// TIA Portal project "Bancada" (V17)

(* hardware
DEVICE "S7-1200 station_1"  S7-1200 Station
   slot 0: "Rack_0"  S7-1200 Rack  Rack  V1.0
   slot 1: "PLC_1"  CPU 1212C AC/DC/Rly  6ES7 212-1BE40-0XB0  V4.5
DEVICE "GSD device_1"  GSD.Device.PN
   slot 0: "Rack"  Rack  V1.0
   slot 0: "danfoss-fc-series"  Danfoss FC PN  130B1135  V03.01.0
      slot 0: "Danfoss FC PN"  Danfoss FC PN
      slot 1: "Interface"  Interface
         slot 1: "Port 1"  Port 1
         slot 2: "Port 2"  Port 2
   slot 1: "PPO 4 - 6/6 Words, Danfoss Telegram 104_1"  PPO 4 - 6/6 Words, Danfoss Telegram 104
      slot 0: "Parameter Access Point"  Parameter Access Point
      slot 1: "PPO 4 - 6/6 Words, Danfoss Telegram 104"  PPO 4 - 6/6 Words, Danfoss Telegram 104
DEVICE "HMI_1"  KTP700 Basic PN
   slot 0: "HMI_1"  KTP700 Basic PN  6AV2 123-2GB03-0AX0  17.0.0.0
   slot 1: "HMI_RT_1"  KTP700 Basic PN  6AV2 123-2GB03-0AX0  17.0.0.0
   slot 5: "HMI_1.IE_CP_1"  PROFINET Interface  17.0.0.0
      slot 1: "PROFINET Interface_1"  PROFINET Interface
         slot 1: "Port_1"  Port
*)

// ===== PLC "PLC_1"  CPU 1212C AC/DC/Rly =====

VAR_GLOBAL   // PLC tag table "teste"
   "Tag_2" AT %M100.0 : Bool;
   "Tag_3" AT %MW300 : Int;
   "Tag_4" AT %MW302 : Int;
   "Tag_5" AT %MW306 : Int;
   "Tag_6" AT %MW308 : Int;
   "Tag_7" AT %MW304 : Int;
   "Tag_8" AT %MW310 : Int;
   "Tag_9" AT %MW312 : Int;
   "Tag_10" AT %MW314 : Int;
   "Tag_11" AT %MW316 : Int;
   "Tag_12" AT %MW320 : Int;
   "Tag_13" AT %MW318 : Int;
   "Tag_14" AT %MD400 : DWord;
   "Tag_15" AT %MD314 : Real;
   "Tag_16" AT %MD318 : Real;
   "Tag_17" AT %MD500 : DWord;
   "Tag_18" AT %MD504 : DWord;
END_VAR

VAR_GLOBAL   // PLC tag table "Default tag table"
   "DRV_EN_DUT1" AT %M0.0 : Bool;
   "RUN_DUT1" AT %M0.1 : Bool;
   "REVERSE_DUT1" AT %M0.2 : Bool;
   "RESET_DUT1" AT %M0.3 : Bool;
   "REF_VALUE_DUT1" AT %MW2 : Int;
   "READY_DUT1" AT %M0.4 : Bool;
   "FAULT_DUT1" AT %M0.5 : Bool;
   "WARNING_DUT1" AT %M0.6 : Bool;
   "RUNNING_DUT1" AT %M0.7 : Bool;
   "RUN_ON_REF_DUT1" AT %M1.0 : Bool;
   "MAV_DUT1" AT %MW4 : Int;
   "MOTORCURRENT_DUT1" AT %MD6 : Real;
   "COMM_ERR_DUT1" AT %MW10 : Int;
   "EXECUTE_DUT1" AT %M1.1 : Bool;
   "RD_WR_DUT1" AT %M1.2 : Bool;
   "PAR_NO_DUT1" AT %MW12 : Word;
   "INDEX_DUT1" AT %MW14 : Word;
   "WR_VALUE_DUT1" AT %MD16 : DWord;
   "BUSY_DUT1" AT %M1.3 : Bool;
   "DONE_DUT1" AT %M1.4 : Bool;
   "FAULT_PARA_DUT1" AT %M1.5 : Bool;
   "RD_VALUE_DUT1" AT %MD20 : DWord;
   "FALUT_CODE_DUT1" AT %MD24 : DWord;
   "CH_ERR_TYP_DUT1" AT %MW28 : Word;
   "ALARM_DUT1" AT %MD30 : DWord;
   "DIAG_WARNING_DUT1" AT %MD34 : DWord;
   "DIAG_ALARM_DUT1" AT %MD38 : DWord;
   "Test" AT %M1.6 : Bool;
   "FB_CTRL_EN_DUT1" AT %M1.7 : Bool;
   "COMM_ERR_FLEXIBLE_DUT1" AT %MW42 : Int;
   "START_FLEXIBLE_CTRL_DUT1" AT %M44.0 : Bool;
   "REF_VALUE_FLEXI_CTRL_DUT1" AT %MW46 : Int;
   "Tag_1" AT %M300.0 : Bool;
   "DC_BRAKE_RAMP" AT %M44.1 : Bool;
   "test1" AT %M44.2 : Bool;
   "Dummy" AT %M44.3 : Bool;
   "PRESET_REF1_DUT1" AT %M44.4 : Bool;
   "PRESET_REF2_DUT1" AT %M44.5 : Bool;
   "DC_BRAKE_RAMP_DUT1" AT %M44.6 : Bool;
   "COAST_INV_DUT1" AT %M44.7 : Bool;
   "QSTP_RMP_DUT1" AT %M45.0 : Bool;
   "HLD_RAMP_DUT1" AT %M45.1 : Bool;
   "RESET_DUT_FLEXIBLE_CTRL_DUT1" AT %M45.2 : Bool;
   "JOG_DUT1" AT %M45.3 : Bool;
   "RAMP_1_2_DUT1" AT %M45.4 : Bool;
   "RLY_1_NO_DUT1" AT %M45.5 : Bool;
   "RLY_2_ON_DUT1" AT %M45.6 : Bool;
   "SETUP_SEL_1_DUT1" AT %M45.7 : Bool;
   "SETUP_SEL_2_DUT1" AT %M48.0 : Bool;
   "REVERSE_FLEXIBLE_CTRl_DUT1" AT %M48.1 : Bool;
   "READ_FLEXIBLE_CTRL_DUT1" AT %M48.2 : Bool;
   "FALUT_FLEXIBLE_CTRL_DUT1" AT %M48.3 : Bool;
   "WARNING_FLEXIBLE_CTRL_DUT1" AT %M48.4 : Bool;
   "RUN_ON_REF_FLEXIBLE_CTRL_DUT1" AT %M48.5 : Bool;
   "RUNNING_FLEXIBLE_CTRL_DUT1" AT %M48.6 : Bool;
   "MAV_FLEXIBLE_CTRL_DUT1" AT %MW50 : Int;
   "EN_BASIC" AT %M48.7 : Bool;
   "EN_FLEXIBLE_CTRL" AT %M49.0 : Bool;
   "EN_FLEXIBLE" AT %M49.1 : Bool;
   "EN_PARAM_ACCESS" AT %M49.2 : Bool;
   "EN_DIAGNOSTICS" AT %M49.3 : Bool;
   "DRV_EN_DUT2" AT %M49.4 : Bool;
   "RUN_DUT2" AT %M49.5 : Bool;
   "REVERSE_DUT2" AT %M49.6 : Bool;
   "RESET_DUT2" AT %M49.7 : Bool;
   "REF_VALUE_DUT2" AT %MW52 : Int;
   "READY_DUT2" AT %M54.0 : Bool;
   "FAULT_DUT2" AT %M54.1 : Bool;
   "WARNING_DUT2" AT %M54.2 : Bool;
   "RUNNING_DUT2" AT %M54.3 : Bool;
   "RUN_ON_REF_DUT2" AT %M54.4 : Bool;
   "MAV_DUT2" AT %MW56 : Int;
   "MOTORCURRENT_DUT2" AT %MD58 : Real;
   "COMM_ERR_DUT2" AT %MW62 : Int;
   "PRESET_REF1_DUT2" AT %M54.5 : Bool;
   "PRESET_REF2_DUT2" AT %M54.6 : Bool;
   "DC_BRAKE_RAMP_DUT2" AT %M54.7 : Bool;
   "COAST_INV_DUT2" AT %M55.0 : Bool;
   "QSTP_RMP_DUT2" AT %M55.1 : Bool;
   "HLD_RAMP_DUT2" AT %M55.2 : Bool;
   "START_FLEXIBLE_CTRL_DUT2" AT %M55.3 : Bool;
   "RESET_DUT_FLEXIBLE_CTRL_DUT2" AT %M55.4 : Bool;
   "JOG_DUT2" AT %M55.5 : Bool;
   "RAMP_1_2_DUT2" AT %M55.6 : Bool;
   "RLY_1_NO_DUT2" AT %M55.7 : Bool;
   "RLY_2_ON_DUT2" AT %M64.0 : Bool;
   "SETUP_SEL_1_DUT2" AT %M64.1 : Bool;
   "SETUP_SEL_2_DUT2" AT %M64.2 : Bool;
   "REVERSE_FLEXIBLE_CTRl_DUT2" AT %M64.3 : Bool;
   "REF_VALUE_FLEXI_CTRL_DUT2" AT %MW66 : Int;
   "READ_FLEXIBLE_CTRL_DUT2" AT %M64.4 : Bool;
   "FALUT_FLEXIBLE_CTRL_DUT2" AT %M64.5 : Bool;
   "WARNING_FLEXIBLE_CTRL_DUT2" AT %M64.6 : Bool;
   "RUNNING_FLEXIBLE_CTRL_DUT2" AT %M64.7 : Bool;
   "MAV_FLEXIBLE_CTRL_DUT2" AT %MW68 : Int;
   "RUN_ON_REF_FLEXIBLE_CTRL_DUT2" AT %M65.0 : Bool;
   "FB_CTRL_EN_DUT2" AT %M65.1 : Bool;
   "COMM_ERR_FLEXIBLE_DUT2" AT %MW70 : Int;
   "DATA_VALID_DUT1" AT %M65.2 : Bool;
   "DATA_VALID_DUT2" AT %M65.3 : Bool;
   "EXECUTE_DUT2" AT %M65.4 : Bool;
   "RD_WR_DUT2" AT %M65.5 : Bool;
   "PAR_NO_DUT2" AT %MW72 : Word;
   "INDEX_DUT2" AT %MW74 : Word;
   "WR_VALUE_DUT2" AT %MD76 : DWord;
   "BUSY_DUT2" AT %M65.6 : Bool;
   "DONE_DUT2" AT %M65.7 : Bool;
   "FAULT_PARA_DUT2" AT %M80.0 : Bool;
   "RD_VALUE_DUT2" AT %MD82 : DWord;
   "FALUT_CODE_DUT2" AT %MD86 : DWord;
   "ALARM_1_DUT1" AT %MD90 : DWord;
   "WARNING_1_DUT1" AT %MD94 : DWord;
   "CH_ERR_TYP_DUT2" AT %MW98 : Word;
   "ALARM_1_DUT2" AT %MD100 : DWord;
   "WARNING_1_DUT2" AT %MD104 : DWord;
END_VAR

VAR_GLOBAL CONSTANT   // PLC tag table "Default tag table"
   "None(1)" : Pip := 65535;
   "Automatic update(1)" : Pip := 0;
   "PIP 1(1)" : Pip := 1;
   "PIP 2(1)" : Pip := 2;
   "PIP 3(1)" : Pip := 3;
   "PIP 4(1)" : Pip := 4;
   "PIP 5" : Pip := 5;
   "PIP 6" : Pip := 6;
   "PIP 7" : Pip := 7;
   "PIP 8" : Pip := 8;
   "PIP 9" : Pip := 9;
   "PIP 10" : Pip := 10;
   "PIP 11" : Pip := 11;
   "PIP 12" : Pip := 12;
   "PIP 13" : Pip := 13;
   "PIP 14" : Pip := 14;
   "PIP 15" : Pip := 15;
   "PIP 16" : Pip := 16;
   "PIP 17" : Pip := 17;
   "PIP 18" : Pip := 18;
   "PIP 19" : Pip := 19;
   "PIP 20" : Pip := 20;
   "PIP 21" : Pip := 21;
   "PIP 22" : Pip := 22;
   "PIP 23" : Pip := 23;
   "PIP 24" : Pip := 24;
   "PIP 25" : Pip := 25;
   "PIP 26" : Pip := 26;
   "PIP 27" : Pip := 27;
   "PIP 28" : Pip := 28;
   "PIP 29" : Pip := 29;
   "PIP 30" : Pip := 30;
   "PIP 31" : Pip := 31;
   "PIP OB Servo(1)" : Pip := 32768;
   "Local~MC(1)" : Hw_SubModule := 51;
   "Local~Display" : Hw_SubModule := 54;
   "Local~Exec(1)" : Hw_SubModule := 52;
   "Local(1)" : Hw_SubModule := 49;
   "Local~DP_interface_1" : Hw_Interface := 60;
   "Local~PROFINET_interface_1(1)" : Hw_Interface := 64;
   "Local~PROFINET_interface_1~Port_1(1)" : Hw_Interface := 65;
   "Local~PROFINET_interface_1~Port_2" : Hw_Interface := 66;
   "Local~PROFINET_interface_2" : Hw_Interface := 72;
   "Local~PROFINET_interface_2~Port_1" : Hw_Interface := 73;
   "OB_Main(1)" : OB_PCYCLE := 1;
   "Local~PROFINET_IO-System" : Hw_IoSystem := 257;
   "OB_Diagnostic error interrupt" : OB_DIAG := 82;
   "Local~DP-Mastersystem" : Hw_IoSystem := 268;
   "profinetdut1~Proxy" : Hw_SubModule := 258;
   "profinetdut1~IODevice" : Hw_Device := 263;
   "profinetdut1~Interface" : Hw_Interface := 259;
   "profinetdut1~Interface~Port_1" : Hw_Interface := 260;
   "profinetdut1~Interface~Port_2" : Hw_Interface := 261;
   "profinetdut1~Head" : Hw_SubModule := 262;
   "profinetdut2~Proxy" : Hw_SubModule := 271;
   "profinetdut2~IODevice" : Hw_Device := 269;
   "profinetdut2~Interface" : Hw_Interface := 272;
   "profinetdut2~Interface~Port_1" : Hw_Interface := 273;
   "profinetdut2~Interface~Port_2" : Hw_Interface := 274;
   "profinetdut2~Head" : Hw_SubModule := 275;
   "Slave_1~Head" : Hw_Interface := 281;
   "Slave_1~DPSlave" : Hw_DpSlave := 279;
   "Slave_1~PPO_Type_2_Module_consistent_PCD_2_1" : Hw_SubModule := 282;
   "Slave_1~PPO_Type_2_Module_consistent_PCD_2_2" : Hw_SubModule := 283;
   "profinetdut1~PPO_4_-_6_6_Words__Danfoss_Telegram,,," : Hw_SubModule := 265;
   "profinetdut1~PPO_4_-_6_6_Words__Danfoss_Telegra,,,~Parameter_Access_Point" : Hw_SubModule := 266;
   "profinetdut1~PPO_4_-_6_6_Words__Danfoss_Telegra,,,~PPO_4_-_6_6_Words__Danfoss_,,," : Hw_SubModule := 267;
   "profinetdut2~PPO_8_-_10_10_Words__Danfoss_Telegr,,," : Hw_SubModule := 276;
   "profinetdut2~PPO_8_-_10_10_Words__Danfoss_Teleg,,,~Parameter_Access_Point" : Hw_SubModule := 277;
   "profinetdut2~PPO_8_-_10_10_Words__Danfoss_Teleg,,,~PPO_8_-_10_10_Words__Danfos,,," : Hw_SubModule := 278;
   "Local~Common(1)" : Hw_SubModule := 50;
   "Local~Device(1)" : Hw_Device := 32;
   "Local~Configuration(1)" : Hw_SubModule := 33;
   "Local~License_Manager" : Hw_SubModule := 42;
   "Local~Virtual_communication_interface" : Hw_Interface := 135;
END_VAR

TYPE "PPO_READ_FCPROFILE"
TITLE = PPO_READ_FCPROFILE
// User defined data tyoe of input data read structure . Holds the data structure obtained from the Process data (PCDREAD) expressed in user data accessible format user
   STRUCT
      STW : Struct   // Status word
         BIT_00_CTRL_RDY : Bool;   // 0=Control not ready, 1=Control ready
         BIT_01_DRV_RDY : Bool;   // 0=Frequency converter, 1=Frequency converter ready
         BIT_02_COAST_RDY : Bool;   // 0=Coasting, 1=Enable
         BIT_03_TRIP : Bool;   // 0=No error, 1=Trip
         BIT_04_ERROR : Bool;   // 0=No error, 1=Error (no trip)
         BIT_05_RESERVED : Bool;   // 0=Reserved, 1=---
         BIT_06_TRIPLOCK : Bool;   // 0=No error, 1=Triplock
         BIT_07_WARNING : Bool;   // 0=No warning, 1=Warning
         BIT_08_RUNNING_REF : Bool;   // 0=Speed <> reference, 1=Speed=reference
         BIT_09_CTRL_SOURCE : Bool;   // 0=Local operation, 1=Bus control
         BIT_10_F_LIMIT_OK : Bool;   // 0=Out of frequency limit, 1=Frequency limit ok
         BIT_11_IN_OPR : Bool;   // 0=No operation, 1=In operation
         BIT_12_IN_AUTOSTART : Bool;   // 0=Frequency converter OK, 1=Stopped, autostart
         BIT_13_VOLT_MAX : Bool;   // 0=Voltage OK, 1=Voltage exceeded
         BIT_14_TORQ_MAX : Bool;   // 0=Torque OK, 1=Torque exceeded
         BIT_15_TIMER_EXD : Bool;   // 0=Timer OK, 1=Timer exceeded
      END_STRUCT;
      MAV : Int;   // Measured Actual Value (Speed) in raw value (-16384) to (+16384)
      PCD_02 : Int;   // Depends on Drive config.
      PCD_03 : Int;   // Depends on Drive config.
      PCD_04 : Int;   // Depends on Drive config.
      PCD_05 : Int;   // Depends on Drive config.
      PCD_06 : Int;   // Depends on Drive config.
      PCD_07 : Int;   // Depends on Drive config.
      PCD_08 : Int;   // Depends on Drive config.
      PCD_09 : Int;   // Depends on Drive config.
   END_STRUCT;
END_TYPE

TYPE "PPO_WRITE_FCPROFILE"
TITLE = PPO_WRITE_FCPROFILE
// User defined data type of input data read structure. Holds the data structure obtained from the Process data(PCDWRITE) expressed in user data accessible format user
   STRUCT
      CTW : Struct   // Control word
         BIT_00_PRESET_REF_1 : Bool;   // 0=Reference value, 1=selection lsb
         BIT_01_PRESET_REF_2 : Bool;   // 0=Reference value, 1=selection msb
         BIT_02_DC_BRAKE_RAMP : Bool := TRUE;   // 0=DC brake, 1=Ramp
         BIT_03_COAST_INV : Bool := TRUE;   // 0=Coasting, 1=No coasting
         BIT_04_QSTP_RMP : Bool := TRUE;   // 0=Quick stop, 1=Ramp
         BIT_05_HLD_RMP : Bool := TRUE;   // 0=Hold output frequency, 1=Use ramp
         BIT_06_START : Bool;   // 0=Ramp stop, 1=Start
         BIT_07_RESET : Bool;   // 0=No function, 1=Reset
         BIT_08_JOG : Bool;   // 0=No function, 1=Jog
         BIT_09_RAMP_1_2 : Bool;   // 0=Ramp 1, 1=Ramp 2
         BIT_10_DATA_VALID : Bool := TRUE;   // 0=Dont use CTW, 1= Use CTW
         BIT_11_RLY_1_ON : Bool := FALSE;   // 0=Relay 01 deactived, 1=Relay 01 active
         BIT_12_RLY_2_ON : Bool := FALSE;   // 0=Relay 02 deactived, 1=Relay 02 active
         BIT_13_SETUP_SEL_1 : Bool := FALSE;   // 0=Parameter set-up, 1=selection lsb
         BIT_14_SETUP_SEL_2 : Bool := FALSE;   // 0=Parameter set-up, 1=selection msb
         BIT_15_REVERSE : Bool;   // 0= No Reverse, 1= Reverse
      END_STRUCT;
      REF_VALUE : Int;   // Main Ref. value (Speed) in raw value. (-16384) to (+16384)
      PCD_02 : Int;   // Depends on Drive config.
      PCD_03 : Int;   // Depends on Drive config.
      PCD_04 : Int;   // Depends on Drive config.
      PCD_05 : Int;   // Depends on Drive config.
      PCD_06 : Int;   // Depends on Drive config.
      PCD_07 : Int;   // Depends on Drive config.
      PCD_08 : Int;   // Depends on Drive config.
      PCD_09 : Int;   // Depends on Drive config.
   END_STRUCT;
END_TYPE

TYPE "PPO_READ_PROFIDRIVE_PROFILE"
   STRUCT
      STW : Struct   // Status word
         BIT_08_RUNNING_REF : Bool;   // 0=Speed <> reference, 1=Speed=reference
         BIT_09_CTRL_SOURCE : Bool;   // 0=Local operation, 1=Bus control
         BIT_10_F_LIMIT_OK : Bool;   // 0=Out of frequency limit, 1=Frequency limit ok
         BIT_11 : Bool;   // Device specific
         BIT_12_IN_AUTOSTART : Bool;   // 0=Frequency converter OK, 1=Stopped, autostart
         BIT_13_DRV_RDY : Bool;   // 0=Drive is not ready, 1=Drive is ready to go to running state
         BIT_14 : Bool;   // ???
         BIT_15 : Bool;   // ???
         BIT_00_CTRL_RDY : Bool;   // 0=Control not ready, 1=Control ready
         BIT_00_RDY_TO_OPR : Bool;   // 0=Not Ready To Operate, 1=Ready To Operate
         BIT_02_OPR_EN : Bool;   // 0=Operation Disabled, 1=Operation Enabled
         BIT_03_FAULT : Bool;   // 0=No Fault, 1=Fault
         BIT_04_COAST_STP : Bool;   // 0=Coast Stop Activated, 1=Coast Stop not Activated
         BIT_05_QUICK_STP : Bool;   // 0=Quick Stop Not Activated, 1=Quick Stop Activated
         BIT_06_SWTCH_ON_INH : Bool;   // 0=Switching On Not Inhibited, 1=Switching On Inhibited
         BIT_07_WARNING : Bool;   // 0=No warning, 1=Warning
      END_STRUCT;
      MAV : Int;   // Main actual value (Speed) in %
      PCD_02 : Int;   // Depends on Drive config.
      PCD_03 : Int;   // Depends on Drive config.
      PCD_04 : Int;   // Depends on Drive config.
      PCD_05 : Int;   // Depends on Drive config.
      PCD_06 : Int;   // Depends on Drive config.
      PCD_07 : Int;   // Depends on Drive config.
      PCD_08 : Int;   // Depends on Drive config.
      PCD_09 : Int;   // Depends on Drive config.
      PCD_11 : Int;   // Depends on Drive config.
   END_STRUCT;
END_TYPE

TYPE "PPO_WRITE_PROFIDRIVE_PROFILE"
   STRUCT
      CTW : Struct   // Control word
         BIT_08_NOTUSED : Bool;   // Not used
         BIT_09_NOTUSED : Bool;   // Not used
         BIT_10_USE_CTRL_WORD : Bool := TRUE;   // 0=No Control by PLC, 1=Control by PLC
         BIT_11_DEV_SPEC : Bool := FALSE;   // Device specific
         BIT_12_DEV_SPEC : Bool := FALSE;   // Device specific
         BIT_13_DEV_SPEC : Bool := FALSE;   // Device specific
         BIT_14_DEV_SPEC : Bool := FALSE;   // Device specific
         BIT_15_DEV_SPEC : Bool;   // Device specific
         BIT_00_ON_1 : Bool;   // 0=Control not ready, 1=Control ready
         BIT_01_COAST_INV : Bool;   // 0=Coast Stop, 1=No Coast Stop
         BIT_02_QUICK_INV : Bool := TRUE;   // 0=Quick Stop, 1=No Quick Stop
         BIT_03_EN_OPR : Bool := TRUE;   // 0=Operation disabled, 1=Operation enabled
         BIT_04_RAMP : Bool := TRUE;   // 0=Reset Ramp Generator, 1=Enable Ramp Generator
         BIT_05_USE_RAMP : Bool := TRUE;   // 0=Freeze Ramp Generator, 1=Unfreeze Ramp Generator
         BIT_06_START : Bool;   // 0=Disable Set Point, 1=Enable Setpoint
         BIT_07_RESET_ERR : Bool;   // 0=No Reset, 1=Reset Fault, rising edge
      END_STRUCT;
      MRV : Int;   // Main Ref. value (Speed) in %
      PCD_02 : Word;   // Depends on Drive config.
      PCD_03 : Word;   // Depends on Drive config.
      PCD_04 : Word;   // Depends on Drive config.
      PCD_05 : Word;   // Depends on Drive config.
      PCD_06 : Word;   // Depends on Drive config.
      PCD_07 : Word;   // Depends on Drive config.
      PCD_08 : Word;   // Depends on Drive config.
      PCD_09 : Word;   // Depends on Drive config.
      PCD_10 : Word;   // Depends on Drive config.
   END_STRUCT;
END_TYPE

TYPE "PPO_DRIVEPROFILE"
   STRUCT
      PPO_PD : Struct
         RD : "PPO_READ_PROFIDRIVE_PROFILE";
         WR : "PPO_WRITE_PROFIDRIVE_PROFILE";
      END_STRUCT;
   END_STRUCT;
END_TYPE

TYPE "PPO_FC"
TITLE = PPO_FC
// User defined data type of Input data read structure and output data write structure. Holds the data structure obtained from the Process data (PCDREAD) and (PCDWRITE) expressed in user data accessible format user
   STRUCT
      PPO_FC : Struct
         RD : "PPO_READ_FCPROFILE";
         WR : "PPO_WRITE_FCPROFILE";
      END_STRUCT;
   END_STRUCT;
END_TYPE

TYPE "PCD"
   STRUCT
      PCD : Struct
         PCDREAD : "PPO_READ_FCPROFILE";
         PCDWRITE : "PPO_WRITE_FCPROFILE";
      END_STRUCT;
   END_STRUCT;
END_TYPE

DATA_BLOCK "VLT_PROFI_FC_DIAGNOSTICS_DB_2"   // DB1
{ S7_Optimized_Access := 'TRUE' }
AUTHOR : Danfoss_Drives
FAMILY : VLT
VERSION : 1.12
// stored: InstanceOfName VLT_PROFI_FC_DIAGNOSTICS
"VLT_PROFI_FC_DIAGNOSTICS"
BEGIN
END_DATA_BLOCK

DATA_BLOCK "VLT_PROFI_FC_PARAM_ACCESS_DB"   // DB2
{ S7_Optimized_Access := 'FALSE' }
AUTHOR : Danfoss
FAMILY : VLT
VERSION : 1.0
// stored: InstanceOfName VLT_PROFI_FC_PARAM_ACCESS
"VLT_PROFI_FC_PARAM_ACCESS"
BEGIN
END_DATA_BLOCK

DATA_BLOCK "VLT_PROFI_FC_DIAGNOSTICS_DB"   // DB3
{ S7_Optimized_Access := 'TRUE' }
AUTHOR : Danfoss
FAMILY : VLT
VERSION : 1.0
// stored: InstanceOfName VLT_PROFI_FC_DIAGNOSTICS
"VLT_PROFI_FC_DIAGNOSTICS"
BEGIN
END_DATA_BLOCK

DATA_BLOCK "VLT_PROFI_FC_FLEXIBLE_CTRL_DB"   // DB5
{ S7_Optimized_Access := 'TRUE' }
AUTHOR : Danfoss
FAMILY : VLT
VERSION : 1.0
// stored: InstanceOfName VLT_PROFI_FC_FLEXIBLE_CTRL
"VLT_PROFI_FC_FLEXIBLE_CTRL"
BEGIN
END_DATA_BLOCK

DATA_BLOCK "VLT_PROFI_FC_PARAM_ACCESS_DB_1"   // DB6
{ S7_Optimized_Access := 'FALSE' }
AUTHOR : Danfoss
FAMILY : VLT
VERSION : 1.0
// stored: InstanceOfName VLT_PROFI_FC_PARAM_ACCESS
"VLT_PROFI_FC_PARAM_ACCESS"
BEGIN
END_DATA_BLOCK

DATA_BLOCK "VLT_PROFI_FC_DIAGNOSTICS_DB_1"   // DB7
{ S7_Optimized_Access := 'TRUE' }
AUTHOR : Danfoss
FAMILY : VLT
VERSION : 1.0
// stored: InstanceOfName VLT_PROFI_FC_DIAGNOSTICS
"VLT_PROFI_FC_DIAGNOSTICS"
BEGIN
END_DATA_BLOCK

DATA_BLOCK "VLT_PROFI_FC_FLEXIBLE_CTRL_DB_1"   // DB8
{ S7_Optimized_Access := 'TRUE' }
AUTHOR : Danfoss
FAMILY : VLT
VERSION : 1.0
// stored: InstanceOfName VLT_PROFI_FC_FLEXIBLE_CTRL
"VLT_PROFI_FC_FLEXIBLE_CTRL"
BEGIN
END_DATA_BLOCK

DATA_BLOCK "data"   // DB9
{ S7_Optimized_Access := 'TRUE' }
VERSION : 0.1
   VAR
      Input2 : Int;
      Input : Int;
   END_VAR
BEGIN
END_DATA_BLOCK

DATA_BLOCK "db2"   // DB10
{ S7_Optimized_Access := 'TRUE' }
VERSION : 0.1
// stored: InstanceOfName web
"web"
BEGIN
END_DATA_BLOCK

DATA_BLOCK "date"   // DB11
{ S7_Optimized_Access := 'TRUE' }
VERSION : 0.1
   VAR
      in : Int;
      corrente : Real;
      frequencia : Real;
      start : Bool;
      reset : Bool;
      reversao : Bool;
      jog : Bool;
   END_VAR
BEGIN
END_DATA_BLOCK

// folder: VLT_PROFI_LIB_V1_12

DATA_BLOCK "VLT_PCD_DATA"   // DB100
TITLE = VLT_PCD_DATA
{ S7_Optimized_Access := 'TRUE' }
AUTHOR : Danfoss_Drives
FAMILY : VLT
VERSION : 1.12
// Data block of input data read structure and output data write structure. Holds the data structure obtained from the Process data (PCDREAD) and (PCDWRITE) expressed in user data accessible format user
   VAR
      VLT_PCD_DATA : Array[0..10] of "PPO_FC";
   END_VAR
BEGIN
END_DATA_BLOCK

// folder: (top level)

FUNCTION_BLOCK "web"   // FB1, LAD
{ S7_Optimized_Access := 'TRUE' }
VERSION : 0.1
   VAR
      timer1 : TON_TIME;
      timer2 : TON_TIME;
   END_VAR
BEGIN

REGION Network 1
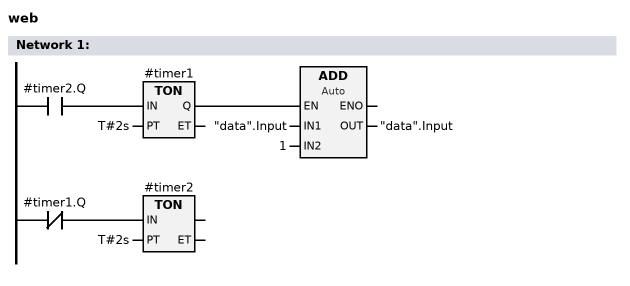
   #timer1(IN := #timer2.Q, PT := T#2s);   // TON
   IF #timer1.Q THEN "data".Input := "data".Input + 1; END_IF;
   #timer2(IN := NOT #timer1.Q, PT := T#2s);   // TON
END_REGION
END_FUNCTION_BLOCK

ORGANIZATION_BLOCK "Main"   // OB1, LAD, ProgramCycle
TITLE = "Main Program Sweep (Cycle)"
{ S7_Optimized_Access := 'TRUE' }
VERSION : 0.1
   VAR_INPUT
      Initial_Call : Bool;   // Initial call of this OB
      Remanence : Bool;   // =True, if remanent data are available
   END_VAR
   VAR_TEMP
      erro : Int;
   END_VAR
   VAR_TEMP   // added for the SCL form of the ladder/FBD networks
      _w1 : Bool;
   END_VAR
BEGIN

REGION Network 1
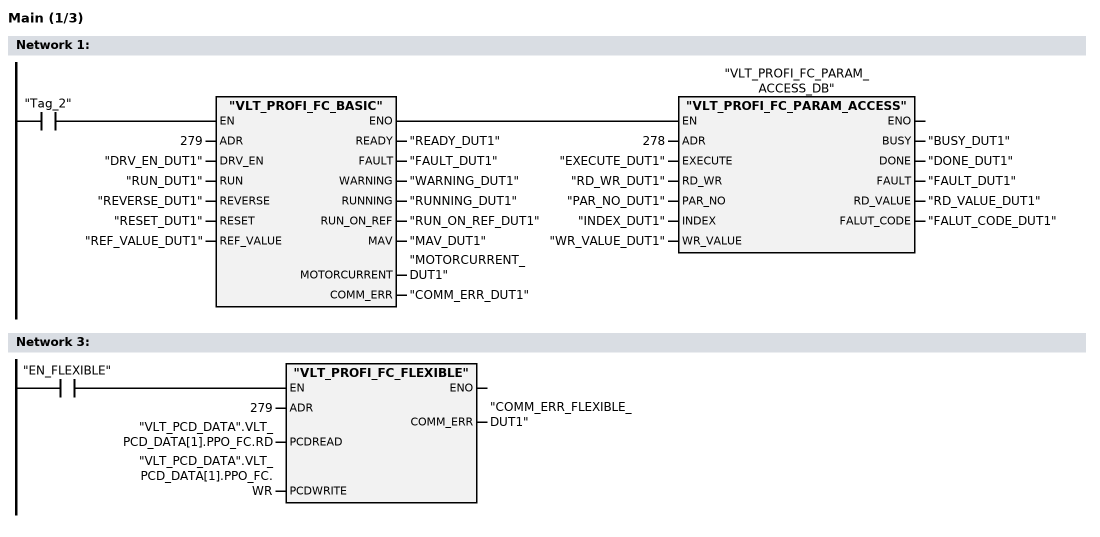
   RUNG wire#powerrail
      Contact( "Tag_2" )
      "VLT_PROFI_FC_BASIC"(ADR := 279, DRV_EN := "DRV_EN_DUT1", RUN := "RUN_DUT1", REVERSE := "REVERSE_DUT1", RESET := "RESET_DUT1", REF_VALUE := "REF_VALUE_DUT1", READY => "READY_DUT1", FAULT => "FAULT_DUT1", WARNING => "WARNING_DUT1", RUNNING => "RUNNING_DUT1", RUN_ON_REF => "RUN_ON_REF_DUT1", MAV => "MAV_DUT1", MOTORCURRENT => "MOTORCURRENT_DUT1", COMM_ERR => "COMM_ERR_DUT1")
      "VLT_PROFI_FC_PARAM_ACCESS_DB"(ADR := 278, EXECUTE := "EXECUTE_DUT1", RD_WR := "RD_WR_DUT1", PAR_NO := "PAR_NO_DUT1", INDEX := "INDEX_DUT1", WR_VALUE := "WR_VALUE_DUT1", BUSY => "BUSY_DUT1", DONE => "DONE_DUT1", FAULT => "FAULT_DUT1", RD_VALUE => "RD_VALUE_DUT1", FALUT_CODE => "FALUT_CODE_DUT1")
   END_RUNG
   // the same network as SCL:
   "VLT_PROFI_FC_BASIC"(EN := "Tag_2",
                        ADR := 279,
                        DRV_EN := "DRV_EN_DUT1",
                        RUN := "RUN_DUT1",
                        REVERSE := "REVERSE_DUT1",
                        RESET := "RESET_DUT1",
                        REF_VALUE := "REF_VALUE_DUT1",
                        READY => "READY_DUT1",
                        FAULT => "FAULT_DUT1",
                        WARNING => "WARNING_DUT1",
                        RUNNING => "RUNNING_DUT1",
                        RUN_ON_REF => "RUN_ON_REF_DUT1",
                        MAV => "MAV_DUT1",
                        MOTORCURRENT => "MOTORCURRENT_DUT1",
                        COMM_ERR => "COMM_ERR_DUT1",
                        ENO => #_w1);
   IF #_w1 THEN
       "VLT_PROFI_FC_PARAM_ACCESS_DB"(ADR := 278,   // "VLT_PROFI_FC_PARAM_ACCESS"
                               EXECUTE := "EXECUTE_DUT1",
                               RD_WR := "RD_WR_DUT1",
                               PAR_NO := "PAR_NO_DUT1",
                               INDEX := "INDEX_DUT1",
                               WR_VALUE := "WR_VALUE_DUT1",
                               BUSY => "BUSY_DUT1",
                               DONE => "DONE_DUT1",
                               FAULT => "FAULT_DUT1",
                               RD_VALUE => "RD_VALUE_DUT1",
                               FALUT_CODE => "FALUT_CODE_DUT1");
   END_IF;
END_REGION

REGION Network 3
   RUNG wire#powerrail
      Contact( "EN_FLEXIBLE" )
      "VLT_PROFI_FC_FLEXIBLE"(ADR := 279, PCDREAD := "VLT_PCD_DATA".VLT_PCD_DATA[1].PPO_FC.RD, PCDWRITE := "VLT_PCD_DATA".VLT_PCD_DATA[1].PPO_FC.WR, COMM_ERR => "COMM_ERR_FLEXIBLE_DUT1")
   END_RUNG
   // the same network as SCL:
   IF "EN_FLEXIBLE" THEN
       "VLT_PROFI_FC_FLEXIBLE"(ADR := 279,
                               PCDREAD := "VLT_PCD_DATA".VLT_PCD_DATA[1].PPO_FC.RD,
                               PCDWRITE := "VLT_PCD_DATA".VLT_PCD_DATA[1].PPO_FC.WR,
                               COMM_ERR => "COMM_ERR_FLEXIBLE_DUT1");
   END_IF;
END_REGION

REGION Network 4
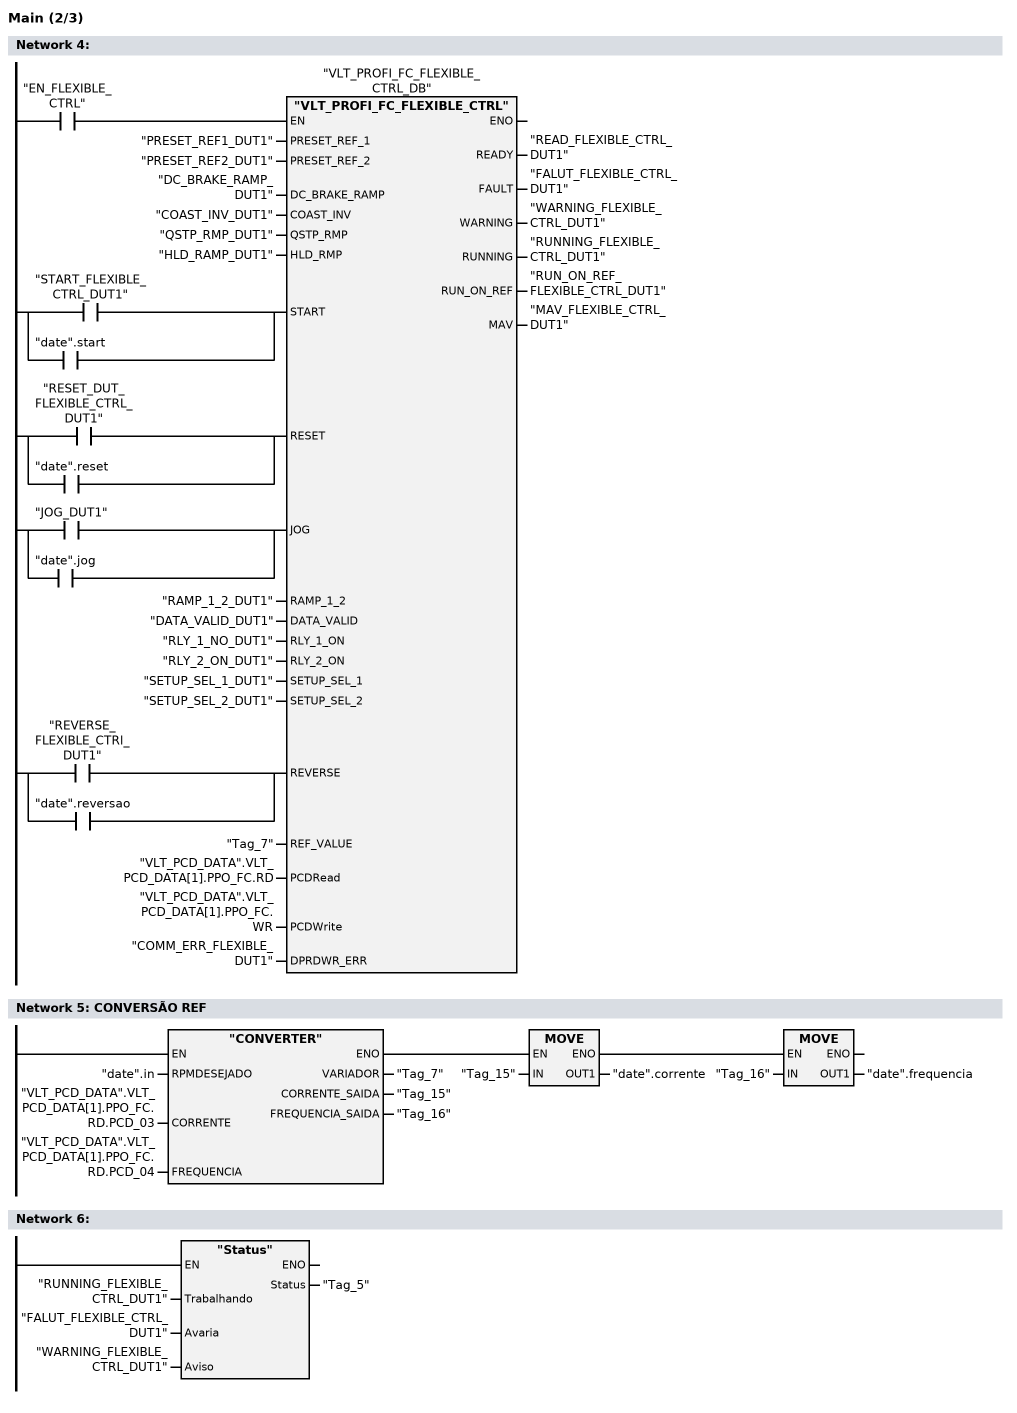
   RUNG wire#powerrail
      Contact( "EN_FLEXIBLE_CTRL" )
      "VLT_PROFI_FC_FLEXIBLE_CTRL_DB"(START := wire#w1, RESET := wire#w2, JOG := wire#w3, REVERSE := wire#w4, PRESET_REF_1 := "PRESET_REF1_DUT1", PRESET_REF_2 := "PRESET_REF2_DUT1", DC_BRAKE_RAMP := "DC_BRAKE_RAMP_DUT1", COAST_INV := "COAST_INV_DUT1", QSTP_RMP := "QSTP_RMP_DUT1", HLD_RMP := "HLD_RAMP_DUT1", RAMP_1_2 := "RAMP_1_2_DUT1", DATA_VALID := "DATA_VALID_DUT1", RLY_1_ON := "RLY_1_NO_DUT1", RLY_2_ON := "RLY_2_ON_DUT1", SETUP_SEL_1 := "SETUP_SEL_1_DUT1", SETUP_SEL_2 := "SETUP_SEL_2_DUT1", REF_VALUE := "Tag_7", PCDRead := "VLT_PCD_DATA".VLT_PCD_DATA[1].PPO_FC.RD, PCDWrite := "VLT_PCD_DATA".VLT_PCD_DATA[1].PPO_FC.WR, DPRDWR_ERR := "COMM_ERR_FLEXIBLE_DUT1", READY => "READ_FLEXIBLE_CTRL_DUT1", FAULT => "FALUT_FLEXIBLE_CTRL_DUT1", WARNING => "WARNING_FLEXIBLE_CTRL_DUT1", RUNNING => "RUNNING_FLEXIBLE_CTRL_DUT1", RUN_ON_REF => "RUN_ON_REF_FLEXIBLE_CTRL_DUT1", MAV => "MAV_FLEXIBLE_CTRL_DUT1")
   END_RUNG
   RUNG wire#powerrail
      Contact( "START_FLEXIBLE_CTRL_DUT1" )
   END_RUNG wire#w1
   RUNG wire#powerrail
      Contact( "date".start )
   END_RUNG wire#w1
   RUNG wire#powerrail
      Contact( "RESET_DUT_FLEXIBLE_CTRL_DUT1" )
   END_RUNG wire#w2
   RUNG wire#powerrail
      Contact( "date".reset )
   END_RUNG wire#w2
   RUNG wire#powerrail
      Contact( "JOG_DUT1" )
   END_RUNG wire#w3
   RUNG wire#powerrail
      Contact( "date".jog )
   END_RUNG wire#w3
   RUNG wire#powerrail
      Contact( "REVERSE_FLEXIBLE_CTRl_DUT1" )
   END_RUNG wire#w4
   RUNG wire#powerrail
      Contact( "date".reversao )
   END_RUNG wire#w4
   // the same network as SCL:
   IF "EN_FLEXIBLE_CTRL" THEN
       "VLT_PROFI_FC_FLEXIBLE_CTRL_DB"(PRESET_REF_1 := "PRESET_REF1_DUT1",   // "VLT_PROFI_FC_FLEXIBLE_CTRL"
                               PRESET_REF_2 := "PRESET_REF2_DUT1",
                               DC_BRAKE_RAMP := "DC_BRAKE_RAMP_DUT1",
                               COAST_INV := "COAST_INV_DUT1",
                               QSTP_RMP := "QSTP_RMP_DUT1",
                               HLD_RMP := "HLD_RAMP_DUT1",
                               START := "START_FLEXIBLE_CTRL_DUT1" OR "date".start,
                               RESET := "RESET_DUT_FLEXIBLE_CTRL_DUT1" OR "date".reset,
                               JOG := "JOG_DUT1" OR "date".jog,
                               RAMP_1_2 := "RAMP_1_2_DUT1",
                               DATA_VALID := "DATA_VALID_DUT1",
                               RLY_1_ON := "RLY_1_NO_DUT1",
                               RLY_2_ON := "RLY_2_ON_DUT1",
                               SETUP_SEL_1 := "SETUP_SEL_1_DUT1",
                               SETUP_SEL_2 := "SETUP_SEL_2_DUT1",
                               REVERSE := "REVERSE_FLEXIBLE_CTRl_DUT1" OR "date".reversao,
                               REF_VALUE := "Tag_7",
                               PCDRead := "VLT_PCD_DATA".VLT_PCD_DATA[1].PPO_FC.RD,
                               PCDWrite := "VLT_PCD_DATA".VLT_PCD_DATA[1].PPO_FC.WR,
                               DPRDWR_ERR := "COMM_ERR_FLEXIBLE_DUT1",
                               READY => "READ_FLEXIBLE_CTRL_DUT1",
                               FAULT => "FALUT_FLEXIBLE_CTRL_DUT1",
                               WARNING => "WARNING_FLEXIBLE_CTRL_DUT1",
                               RUNNING => "RUNNING_FLEXIBLE_CTRL_DUT1",
                               RUN_ON_REF => "RUN_ON_REF_FLEXIBLE_CTRL_DUT1",
                               MAV => "MAV_FLEXIBLE_CTRL_DUT1");
   END_IF;
END_REGION

REGION Network 5: CONVERSÃO REF
   RUNG wire#powerrail
      "CONVERTER"(RPMDESEJADO := "date".in, CORRENTE := "VLT_PCD_DATA".VLT_PCD_DATA[1].PPO_FC.RD.PCD_03, FREQUENCIA := "VLT_PCD_DATA".VLT_PCD_DATA[1].PPO_FC.RD.PCD_04, VARIADOR => "Tag_7", CORRENTE_SAIDA => "Tag_15", FREQUENCIA_SAIDA => "Tag_16")
      Move(in := "Tag_15", out1 => "date".corrente)
      Move(in := "Tag_16", out1 => "date".frequencia)
   END_RUNG
   // the same network as SCL:
   "CONVERTER"(RPMDESEJADO := "date".in,
               CORRENTE := "VLT_PCD_DATA".VLT_PCD_DATA[1].PPO_FC.RD.PCD_03,
               FREQUENCIA := "VLT_PCD_DATA".VLT_PCD_DATA[1].PPO_FC.RD.PCD_04,
               VARIADOR => "Tag_7",
               CORRENTE_SAIDA => "Tag_15",
               FREQUENCIA_SAIDA => "Tag_16",
               ENO => #_w1);
   IF #_w1 THEN
       "date".corrente := "Tag_15";
       "date".frequencia := "Tag_16";
   END_IF;
END_REGION

REGION Network 6
   RUNG wire#powerrail
      "Status"(Trabalhando := "RUNNING_FLEXIBLE_CTRL_DUT1", Avaria := "FALUT_FLEXIBLE_CTRL_DUT1", Aviso := "WARNING_FLEXIBLE_CTRL_DUT1", Status => "Tag_5")
   END_RUNG
   // the same network as SCL:
   "Status"(Trabalhando := "RUNNING_FLEXIBLE_CTRL_DUT1",
            Avaria := "FALUT_FLEXIBLE_CTRL_DUT1",
            Aviso := "WARNING_FLEXIBLE_CTRL_DUT1",
            Status => "Tag_5");
END_REGION

REGION Network 7
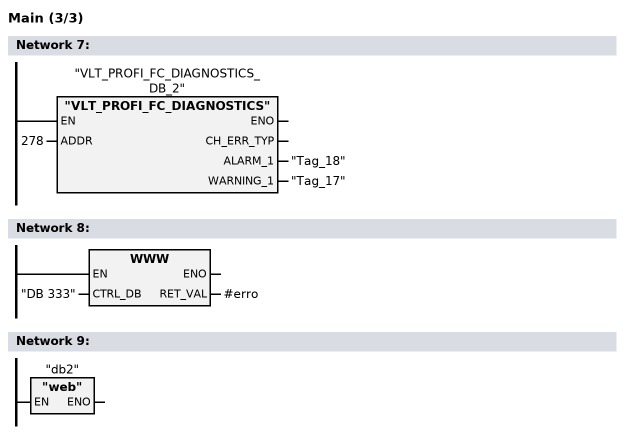
   RUNG wire#powerrail
      "VLT_PROFI_FC_DIAGNOSTICS_DB_2"(ADDR := 278, CH_ERR_TYP =>, ALARM_1 => "Tag_18", WARNING_1 => "Tag_17")
   END_RUNG
   // the same network as SCL:
   "VLT_PROFI_FC_DIAGNOSTICS_DB_2"(ADDR := 278, ALARM_1 => "Tag_18", WARNING_1 => "Tag_17");   // "VLT_PROFI_FC_DIAGNOSTICS"
END_REGION

REGION Network 8
   #erro := WWW(CTRL_DB := "DB 333");
END_REGION

REGION Network 9
   RUNG wire#powerrail
      "db2"()
   END_RUNG
   // the same network as SCL:
   "db2"();   // "web"
END_REGION
END_ORGANIZATION_BLOCK

// folder: VLT_PROFI_LIB_V1_12

FUNCTION_BLOCK "VLT_PROFI_FC_PARAM_ACCESS"   // FB300, SCL
TITLE = VLT_PROFI_FC_PARAM_ACCESS
{ S7_Optimized_Access := 'FALSE' }
AUTHOR : Danfoss_Drives
FAMILY : VLT
VERSION : 1.12
// Parameter Access Functio Block
   VAR_INPUT
      ADR : Hw_Io;   // S7-1200/1500 requires HW Identifier. Can be found in HW configuration for the specific PPO type
      EXECUTE : Bool;   // 1 = The rising edge of this signal starts the requested operation, 0 = Triggers an ACK of the end-of-operation notification and the client is
      RD_WR : Bool;   // 0= Parameter read operation , 1= Parameter write operation
      PAR_NO : Word;   // Enter the drive parameter number in the Hex format. (Example :Parameter -341=155Hex) (Ramp1 Ramp Up Time)
      INDEX : Word;   // Enter the index number (Example: Parameter 310 [2]) 310-Parameter number and 2-Index number
      WR_VALUE : DWord;   // Write value to the drive
   END_VAR
   VAR_OUTPUT
      BUSY : Bool;   // 0= Execution is not started or execution is completed , 1= Execution is processing
      DONE : Bool;   // 0= Value exchange is not completed, 1= Value exchange is completed
      FAULT : Bool;   // 0= Value exchange is completed, 1= Value exchange is unsuccessful.
      RD_VALUE : DWord;   // Read value from the drive
      FALUT_CODE : DWord;   // Indicates the error code associated with the most recently executed command.
   END_VAR
   VAR
      Request_rec : Struct   // Request record
         Req_Header : Struct
            Request_Ref : Byte;
            Request_ID : Byte;
            Axis_Number : Byte;
            No_of_Parameter : Byte;
         END_STRUCT;
         Req_ParaAddress : Struct
            Attribute : Byte;
            Num_of_elements : Byte;
            Parameter_Num : Word;
            Subindex : Word;
            Write_Format : Byte;
            Write_Num_Of_Value : Byte;
            Write_Value : Array[1..4] of Byte;
         END_STRUCT;
      END_STRUCT;
      Response_rec : Struct   // Response record
         Res_Header : Struct
            Reqest_Ref : Byte;
            Request_ID : Byte;
            Axis_Number : Byte;
            No_Of_Parameter : Byte;
         END_STRUCT;
         Res_Data : Array[1..6] of Byte;
      END_STRUCT;
      WRREC_Instance : WRREC;   // Write record instance
      RDREC_Instance : RDREC;   // Read record instance
      Response_Len : UInt;   // Response length
      Case_sequence_selection : Int;   // Case sequence selection
      Static_fault : Bool;   // Read fault status
      Static_done : Bool;   // Done status
      Static_busy : Bool;   // Busy status
      Static_valid : Bool;   // Valid status
      Static_bool_1 : Bool;   // Static bit of read start enble
      Static_bool_2 : Bool;   // Static bit of write start enble
      Static_bool_3 : Bool;   // Static bit of NOT RD_WR
      Static_bool_4 : Bool;   // Static bit of write done
      Static_bool_5 : Bool;   // Static bit of Capturing the falling edge of Last value
      Static_bool_6 : Bool;   // Static bit of start write request
      Static_stored_status : DWord;   // Stored status of error code
   END_VAR
   VAR_TEMP
      Temp_word_high : Word;   // Word high
      Temp_word_low : Word;   // Word low
      Temp_word1 : Word;   // Dword input to high word
      Temp_word2 : Word;   // Dword input to low word
      Temp_dword_high : DWord;   // Double word high
      Temp_dword_low : DWord;   // Double word low
   END_VAR
BEGIN
   //-------------------------------------------------------------------------------------------------------------
   // VLT_PROFI_FC_PARAM_ACCESS: Rev. V1.12
   // Valid for S7-1200 and S7-1500 Type CPU's.
   // Block handles communication with a VLT frequency converter. Either Trough PROFINET OR PROFIBUS.
   // Acyclic communication with VLT.
   // Can be done in HW config of S7, on the Drive LCP or MCT10.
   //-------------------------------------------------------------------------------------------------------------

       #Static_bool_3 := NOT #RD_WR;                                              // Static bit is NOT of RD_WR

   // Initializing the value with Zero
       IF (#EXECUTE AND NOT #Static_bool_5) THEN
       #DONE := 0;
       #BUSY := 0;
       #FAULT := 0;
       #FALUT_CODE := 0;
       #Static_busy := 0;
       #Static_done := 0;
       #Static_fault := 0;
       FILL_BLK(IN := 0,
                COUNT := 6,
               OUT => #Response_rec.Res_Data[1]);     // Read array initializing the value with Zero
       END_IF;

       //Parameter Read Value Operation Enable
       IF (#Static_bool_3) AND (#EXECUTE AND NOT #Static_bool_5) THEN                    //Read with rising edge command
       #Case_sequence_selection := 11;                                         //Case sequence selection
       #RD_VALUE := 0;                                                         //Read value to zero
       #Static_bool_1 := 1;                                                       //Start request enable

       //Parameter Write Value Operation Enable
       ELSIF (#RD_WR) AND (#EXECUTE AND NOT #Static_bool_5) THEN                      //Write with rising edge command
       #Case_sequence_selection := 11;                                         //Case sequence selection
       #RD_VALUE := 0;                                                         //Read value to zero
       #Static_bool_2 := 1;                                                       //Start request enable
       END_IF;

       //Read or Write request parameter values are generally transferred via the header of the RECORD data record
       #Request_rec.Req_Header.Request_Ref := B#16#01;                            //Request reference 
       #Request_rec.Req_Header.Axis_Number := B#16#00;                            //Axis number
       #Request_rec.Req_Header.No_of_Parameter := B#16#01;                        //Number of parameter
       #Request_rec.Req_ParaAddress.Attribute := B#16#10;                         //Attribute
       #Request_rec.Req_ParaAddress.Num_of_elements := B#16#01;                   //Number of element
       #Request_rec.Req_ParaAddress.Parameter_Num := (#PAR_NO);                   //Parameter number
       #Request_rec.Req_ParaAddress.Subindex := #INDEX;                           //Sub index

       //Read Request parameter values are generally transferred via the header of the RECORD data record
       IF #Static_bool_1 THEN
       #Request_rec.Req_Header.Request_ID := 16#51;                               //Read request, 51=Read request, Dword format
       END_IF;

       // Write Request request parameter values are generally transferred via the header of the RECORD data record
       IF #Static_bool_2 THEN
       #Request_rec.Req_Header.Request_ID := B#16#52;                            //Change request, 52=Write request, Dword format
       #Request_rec.Req_ParaAddress.Write_Format := B#16#43;                     //Write format
       #Request_rec.Req_ParaAddress.Write_Num_Of_Value := B#16#01;               //Write number of value

       //Write value
       #Request_rec.Req_ParaAddress.Write_Value[4] := WORD_TO_BYTE(DWORD_TO_WORD(#WR_VALUE));
       #Request_rec.Req_ParaAddress.Write_Value[3] := WORD_TO_BYTE(DWORD_TO_WORD(SHR(IN := (#WR_VALUE), N := 8)));
       #Request_rec.Req_ParaAddress.Write_Value[2] := WORD_TO_BYTE(DWORD_TO_WORD(SHR(IN := (#WR_VALUE), N := 16)));
       #Request_rec.Req_ParaAddress.Write_Value[1] := WORD_TO_BYTE(DWORD_TO_WORD(SHR(IN := (#WR_VALUE), N := 24)));
       END_IF;

       CASE #Case_sequence_selection OF
       11:  // Statement section case 11
       IF (#Static_bool_1 OR #Static_bool_2)  THEN
               #Static_bool_6 := 1;
               #BUSY := 1;
       END_IF;
       ;
       IF #Static_bool_6 AND NOT #Static_done THEN   //Start WRREC request 
           #WRREC_Instance(REQ := TRUE,           //WRREC Instance                        
                       ID := #ADR,
                       INDEX := 47,
                       BUSY => #Static_busy,
                       DONE => #Static_done,
                       ERROR => #Static_fault,
                       LEN := 16,
                       RECORD := #Request_rec,
                       STATUS => #Static_stored_status);
       END_IF;
       ;
       IF #Static_done OR #Static_fault AND NOT #Static_busy THEN     //Write request status, done or fault or busy
       #Case_sequence_selection := 12;      //12 Case sequence selection
       END_IF;
       ;
       12: // Statement section case 12
       IF #Static_done = 1 THEN                    //Check parameter write is done 
          #Case_sequence_selection := 13;          //13 Case sequence selection
          #DONE := 0;
          #BUSY := 1;
          #Static_bool_4 := 1;
          ;
   ELSIF #Static_fault = 1 THEN               //Check write record is fault
         #Case_sequence_selection := 50;      //50 Case sequence selection
         #FAULT := 1;
         #BUSY := 0;
         #FALUT_CODE := (#Static_stored_status);     //Fault code value
     END_IF;
     ;
       13: // Statement section case 13
       IF #Static_bool_4 AND (NOT #Static_valid) THEN   //Start RDREC response 
       #RDREC_Instance(REQ := TRUE,            //RDREC Instance
                        ID := #ADR,
                        INDEX := 47,
                        MLEN := 10,
                        BUSY => #Static_busy,
                        LEN => #Response_Len,
                        STATUS => #Static_stored_status,
                        VALID => #Static_valid,
                        RECORD := #Response_rec);
       END_IF;
       ;
   IF #Static_valid = 1 AND #Static_bool_3 THEN    //Read response is valid
    IF #Response_rec.Res_Data[1] = 16#44 OR #Response_rec.Res_Header.Request_ID = 16#D1 THEN   //Check the parameter format
       #FAULT := 1;
       #DONE := 0;
       #BUSY := 0;
       #Case_sequence_selection := 60; //Fault State
       #RD_VALUE := 0;
       ;
     ELSE
       #FAULT := 0;
       #DONE := 1;
       #BUSY := 0;
       #Case_sequence_selection := 14; //Done State

       END_IF;
             ;
   ELSIF #Static_busy = 1 THEN     //Busy State
         #Case_sequence_selection := 13;
         #BUSY := 1;
       END_IF;
             ;
    IF #Static_valid = 1 AND #RD_WR THEN
     IF #Response_rec.Res_Data[1] = 16#44 OR #Response_rec.Res_Header.Request_ID = 16#82 THEN  // Statement section IF
        #FAULT := 1;
        #DONE := 0;
        #BUSY := 0;
        #Case_sequence_selection := 60; //Fault State
        #RD_VALUE := 0;

       ELSE
        #FAULT := 0;
        #DONE := 1;
        #BUSY := 0;
        #Case_sequence_selection := 15; //Done State
       END_IF;
             ;
   ELSIF #Static_busy = 1 THEN     //Busy State
         #Case_sequence_selection := 13;
         #BUSY := 1;
       END_IF;
             ;
       14: // Statement section case 14
           // Parameter Read done state
           #DONE := 1;
           #BUSY := 0;
           #FALUT_CODE := 16#FF;       //If error is not present in the read or write operation and then error code is set as 0xFF. Since 0x00 is valid error code for Unknown Parameter.

           // Read value is converted from Word to DWord
           #Temp_word_high := SHL(IN := BYTE_TO_WORD(#Response_rec.Res_Data[3]), N := 8);
           #Temp_word_low := BYTE_TO_WORD(#Response_rec.Res_Data[4]);
           #Temp_word1 := #Temp_word_high XOR #Temp_word_low;

           #Temp_word_high := SHL(IN := BYTE_TO_WORD(#Response_rec.Res_Data[5]), N := 8);
           #Temp_word_low := BYTE_TO_WORD(#Response_rec.Res_Data[6]);
           #Temp_word2 := #Temp_word_high XOR #Temp_word_low;

           #Temp_dword_high := SHL(IN := WORD_TO_DWORD(#Temp_word1), N := 16);
           #Temp_dword_low := WORD_TO_DWORD(#Temp_word2);
           #RD_VALUE := (#Temp_dword_high XOR #Temp_dword_low); //Read Value
           ;
       15: // Statement section case 15
           // Parameter Write done state
           #DONE := 1;
           #BUSY := 0;
           #FALUT_CODE := 16#FF;       //If error is not present in the read or write operation and then error code is set as 0xFF. Since 0x00 is valid error code for Unknown Parameter.
           ;
       50: // Statement section case 50
           // Parameter write Fault state 
           #FAULT := 1;                         //Fault status
           #DONE := 0;
           #BUSY := 0;
           #FALUT_CODE := (#Static_stored_status);      //Fault code value
           ;
       60: // Statement section case 60
           // Parameter Response error state
           #FAULT := 1;                         //Fault status
           #DONE := 0;
           #BUSY := 0;
           #Temp_word_high := SHL(IN := BYTE_TO_WORD(#Response_rec.Res_Data[3]), N := 8);
           #Temp_word_low := BYTE_TO_WORD(#Response_rec.Res_Data[4]);
           #FALUT_CODE := #Temp_word_high XOR #Temp_word_low;      //Fault code moving to stored status
           ;
       END_CASE;

       IF NOT #EXECUTE THEN            // If execute command is not present then zero value moved to below variables
          #Static_bool_1 := 0;
          #Static_bool_2 := 0;
          #Static_bool_4 := 0;
          #Static_bool_6 := 0;
          #Static_valid := 0;
       END_IF;
             ;
           #Static_bool_5 := #EXECUTE;        //Capturing the falling edge of Last value
END_FUNCTION_BLOCK

FUNCTION_BLOCK "VLT_PROFI_FC_FLEXIBLE_CTRL"   // FB301, SCL
TITLE = VLT_PROFI_FC_FLEXIBLE_CTRL
{ S7_Optimized_Access := 'TRUE' }
AUTHOR : Danfoss_Drives
FAMILY : VLT
VERSION : 1.12
// Flexible Control Function Block
   VAR_INPUT
      PRESET_REF_1 : Bool;   // Bit 0. 0=Reference value, 1=selection lsb
      PRESET_REF_2 : Bool;   // Bit 1. 0=Reference value, 1=selection msb
      DC_BRAKE_RAMP : Bool := TRUE;   // Bit 2. 0=DC brake, 1=Ramp
      COAST_INV : Bool := TRUE;   // Bit 3. 0=Coasting, 1=No coasting
      QSTP_RMP : Bool := TRUE;   // Bit 4. 0=Quick stop, 1=Ramp
      HLD_RMP : Bool := TRUE;   // Bit 5. 0=Hold output frequency, 1=Use ramp
      START : Bool;   // Bit 6. 0=Ramp stop, 1=Start
      RESET : Bool;   // Bit 7. 0=No function, 1=Reset
      JOG : Bool;   // Bit 8. 0=No function, 1=Jog
      RAMP_1_2 : Bool;   // Bit 9. 0=Ramp 1, 1=Ramp 2
      DATA_VALID : Bool := TRUE;   // Bit 10. 0=Dont use CTW, 1=Use CTW
      RLY_1_ON : Bool := FALSE;   // Bit 11. 0=Relay 01 deactived, 1=Relay 01 active
      RLY_2_ON : Bool := FALSE;   // Bit 12. 0=Relay 02 deactived, 1=Relay 02 active
      SETUP_SEL_1 : Bool := FALSE;   // Bit 13. 0=Parameter set-up, 1=selection lsb. Multi setup in P. 0-10 must be selected.
      SETUP_SEL_2 : Bool := FALSE;   // Bit 14. 0=Parameter set-up, 1=selection msb. Multi setup in P. 0-10 must be selected.
      REVERSE : Bool;   // Bit 15. 0= No Reverse, 1= Reverse
      REF_VALUE : Int;   // Main Ref. value (Speed) in raw value. (-16384) to (+16384)
   END_VAR
   VAR_OUTPUT
      READY : Bool;   // Drive ready to start
      FAULT : Bool;   // Fault is present. Trip or Trip lock
      WARNING : Bool;   // Warning present
      RUNNING : Bool;   // Drive is started but not necessarily running on reference speed.
      RUN_ON_REF : Bool;   // Running on reference
      MAV : Int;   // Measured Actual Value (Speed) in raw value (-16384) to (+16384)
   END_VAR
   VAR_IN_OUT
      PCDRead : "PPO_READ_FCPROFILE";   // Pointer to data structure for FC data
      PCDWrite : "PPO_WRITE_FCPROFILE";   // Pointer to data structure for FC data
      DPRDWR_ERR : Int;   // Map the COMM_ERR tag from VLT_PROFI_FC_FLEXIBLE Function Block
   END_VAR
BEGIN
   //-------------------------------------------------------------------------------------------------------------
   // VLT_PROFI_FC_FLEXIBLE_CTRL: Rev. V1.12
   // Valid for S7-1200 and S7-1500 Type CPU's.
   // This FB is to be used together with "VLT_PROFI_FC_FLEXIBLE"
   // This FB is designed to work with the FCPROFILE on the VLT which is the default setting.
   // Block Manages control and status bits' as well as Reference value. The default values on the Input Interface definitions
   // are set as if they are not assigned an outside value, it will bring the VLT in a "Ready to Start" State.
   //-------------------------------------------------------------------------------------------------------------


   //------------------------------------Settings of Controlword--------------------------------------------------
   // Prepare all Controlword Bit's to default values so that
   // they are in a "ready to start" mode. CTW =043Ch
   #PCDWrite.CTW.BIT_00_PRESET_REF_1 := #PRESET_REF_1;
   #PCDWrite.CTW.BIT_01_PRESET_REF_2 := #PRESET_REF_2;
   #PCDWrite.CTW.BIT_02_DC_BRAKE_RAMP := #DC_BRAKE_RAMP;
   #PCDWrite.CTW.BIT_03_COAST_INV := #COAST_INV;
   #PCDWrite.CTW.BIT_04_QSTP_RMP := #QSTP_RMP;
   #PCDWrite.CTW.BIT_05_HLD_RMP := #HLD_RMP;
   #PCDWrite.CTW.BIT_06_START := #START;
   #PCDWrite.CTW.BIT_07_RESET := #RESET;
   #PCDWrite.CTW.BIT_08_JOG := #JOG;
   #PCDWrite.CTW.BIT_09_RAMP_1_2 := #RAMP_1_2;
   #PCDWrite.CTW.BIT_10_DATA_VALID := #DATA_VALID;
   #PCDWrite.CTW.BIT_11_RLY_1_ON := #RLY_1_ON;
   #PCDWrite.CTW.BIT_12_RLY_2_ON := #RLY_2_ON;
   #PCDWrite.CTW.BIT_13_SETUP_SEL_1 := #SETUP_SEL_1; //  Multi setup in P. 0-10 must be selected.
   #PCDWrite.CTW.BIT_14_SETUP_SEL_2 := #SETUP_SEL_2; //  Multi setup in P. 0-10 must be selected.
   #PCDWrite.CTW.BIT_15_REVERSE := #REVERSE;
   //------------------------------------Settings of Controlword---------------------------------------------------

   //------------------------------------Set reference speed-------------------------------------------------------
   #PCDWrite.REF_VALUE := #REF_VALUE; // Reference speed is a RAW value - 16384 to + 16384.
   //------------------------------------Set reference speed-------------------------------------------------------

   //------------------------------------Mask out Drive status bit's-----------------------------------------------
   // These are those considered to be used most often, there fore put in as "OUTPUT's" on the FB.
   #READY := (#PCDRead.STW.BIT_00_CTRL_RDY AND #PCDRead.STW.BIT_01_DRV_RDY AND #PCDRead.STW.BIT_02_COAST_RDY AND #PCDRead.STW.BIT_09_CTRL_SOURCE); // Drive ready to start from Fieldbus
   #RUNNING := #PCDRead.STW.BIT_11_IN_OPR; // Drive is started but not necessarily running on reference speed.
   #RUN_ON_REF := #PCDRead.STW.BIT_08_RUNNING_REF; // Running on reference
   #WARNING := #PCDRead.STW.BIT_07_WARNING; // Warning present
   #FAULT := (#PCDRead.STW.BIT_04_ERROR OR #PCDRead.STW.BIT_03_TRIP OR #PCDRead.STW.BIT_06_TRIPLOCK); // Fault present. Trip or Trip lock
   //------------------------------------Mask out Drive status bit's-----------------------------------------------

   //------------------------------------Extraction of Main actual value--------------------------------------------
   #MAV := #PCDRead.MAV; // Main Actual Value(MAV) is read from the Drive as - 16384 to + 16384. 
   //------------------------------------Extraction of Main actual value--------------------------------------------

   //------------------------------------Initialize input's to their default values--------------------------------
   // This set's the default values for the input definitions. This ensures that if an input is not configured.
   // it will always have it initial default value
   #PRESET_REF_1 := FALSE;
   #PRESET_REF_2 := FALSE;
   #DC_BRAKE_RAMP := TRUE;
   #COAST_INV := TRUE;
   #QSTP_RMP := TRUE;
   #HLD_RMP := TRUE;
   #START := FALSE;
   #RESET := FALSE;
   #JOG := FALSE;
   #RAMP_1_2 := FALSE;
   #RLY_1_ON := FALSE;
   #RLY_2_ON := FALSE;
   #SETUP_SEL_1 := FALSE;
   #SETUP_SEL_2 := FALSE;
   #REVERSE := FALSE;
   #DATA_VALID := TRUE;
   //------------------------------------Initialize input's to their default values--------------------------------

   //------------------------------------Ensure ENO is TRUE always--------------------------------------------------
   ENO := TRUE;
   //------------------------------------Ensure ENO is TRUE always--------------------------------------------------
END_FUNCTION_BLOCK

FUNCTION_BLOCK "VLT_PROFI_FC_DIAGNOSTICS"   // FB302, SCL
TITLE = VLT_PROFI_FC_DIAGNOSTICS
{ S7_Optimized_Access := 'TRUE' }
AUTHOR : Danfoss_Drives
FAMILY : VLT
VERSION : 1.12
// Diagnostics Function Block
   VAR_INPUT
      ADDR : Hw_Io;   // S7-1200/1500 requires HW Identifier. Can be found in HW configuration for the specific PPO type
   END_VAR
   VAR_OUTPUT
      CH_ERR_TYP : Word;   // Channel Number Error Type
      ALARM_1 : DWord;   // Alarm is present (Profibus or Profinet)
      WARNING_1 : DWord;   // Warning present (Profibus or Profinet)
   END_VAR
   VAR
      RALRM_Instance : RALRM;   // RALARM Instance
      Static_1 : Struct   // Static memory tags
         AlarmMode : Int := 2;   // Alarm mode
         AlarmCheckID : Hw_Io := 0;   // S7-1200/1500 requires HW Identifier. Can be found in HW configuration for the specific PPO type
         AlarmStatus : DWord;   // Error code
         AlarmFromID : Hw_Io;   // Hardware mirror ID
         AlarmReceived : Bool;   // New interrupt was received
         AlarmMaxLength : UInt;   // Maximum length of the interrupt information to be received in bytes
         AlarmLength : UInt;   // Length of the received interrupt information
         TI_DiagnosticInterrupt : TI_DiagnosticInterrupt;
         Additional_Diag : Struct   // Not used
            Header : Struct
               BlockType : Word;
               BlockLength : UInt;
               "Version" : Word;
               InterruptType : UInt;
               API : DWord;
               SlotNumber : UInt;
               SubSlotNumber : UInt;
               ModulSpecInfo : DWord;
               SubModulSpecInfo : DWord;
               InterruptSpecifier : DWord;
            END_STRUCT;
            addInfo : Struct
               FormatIdentifier : Word;
               ChannelNumber : Word;
               ChannelErrorType : Byte;
               DataFormat : Byte;
               ErrorCode : Word;
            END_STRUCT;
         END_STRUCT;
      END_STRUCT;
      AINFOManufacture : Struct   // ANIFO Manufature
         W0_block_type : Word;   // Block type
         W2_block_length : Word;   // Block length
         W4_version : Word;   // Version
         W6_interrupt_type : Word;   // ID for interrupt type:Diagnostics interrupt (incoming or outgoing)
         D8_API : DWord;   // API (Application Process Identifier)
         W12_comp_slot_num : Word;   // Slot number of the component triggering the interrupt
         W14_submodule_slot_num : Word;   // Submodule slot number of the component triggering the interrupt
         D16_module_ID : DWord;   // Module identification; specific information on the source of the interrupt
         D20_submodule_ID : DWord;   // Submodule identification; specific information on the source of the interrupt
         W24_interrupt_specifer : Word;   // Interrupt specifier
         W26_Add_W0_format_ID : Word;   // ID format
         D28_AlarmWord : DWord;   // Profibus Alarm word
         D32_WarnWord : DWord;   // Profibus Warning word
         D36_PdriveWarnWord : DWord;   // Profidrive warning word
         D38_extended_info : DWord;   // Extended information
      END_STRUCT;
      SlaveType : Int;   // Slave type (Profibus or Profinet)
      ProfibusAlarm : DWord;   // ProfibusAlarm
      ProfibusWarning : DWord;   // ProfibusWarning
      TempAlarm : DWord;   // Temporary alarm receive
      TempWarning : DWord;   // Temporary warning receive
      Profibus_slave : Bool;   // Profibus slave
      Profinet_slave : Bool;   // Profinet slave
   END_VAR
   // // Static_1.TI_DiagnosticInterrupt.SI_Format : Format of the start information
   // // Static_1.TI_DiagnosticInterrupt.OB_Class : OB Class
   // // Static_1.TI_DiagnosticInterrupt.OB_Nr : OB Number
   // // Static_1.TI_DiagnosticInterrupt.LADDR : Hardware address of the component triggering the interrupt
   // // Static_1.TI_DiagnosticInterrupt.IO_State : Slot number of the component triggering the interrupt
   // // Static_1.TI_DiagnosticInterrupt.address : Address information
   // // Static_1.TI_DiagnosticInterrupt.slv_prfl : Slave profile( Profinet or Profibus)
   // // Static_1.TI_DiagnosticInterrupt.intr_type : Interrupt info type
   // // Static_1.TI_DiagnosticInterrupt.flags1 : Flags of the PROFIBUS DP master interface module / PROFINET IO controller interface module
   // // Static_1.TI_DiagnosticInterrupt.flags2 : Flags of the PROFIBUS DP master interface module / PROFINET IO controller interface module
   // // Static_1.TI_DiagnosticInterrupt.id : Management information
   // // Static_1.TI_DiagnosticInterrupt.manufacturer : Manufacturer ID (only in a distributed configuration with PROFINET IO).
   // // Static_1.TI_DiagnosticInterrupt.instance : Ident number of the instance (only in a distributed configuration with PROFINET IO).
   // // Static_1.TI_DiagnosticInterrupt.MultiError : Error code
   // // Static_1.TI_DiagnosticInterrupt.Channel : Chennal
BEGIN


   #Static_1.AlarmCheckID := #ADDR;                         



   "RALRM_DB"(MODE := #Static_1.AlarmMode,                   
              F_ID := #Static_1.AlarmCheckID,                
              MLEN := #Static_1.AlarmMaxLength,             
              NEW => #Static_1.AlarmReceived,               
              STATUS => #Static_1.AlarmStatus,               
              ID => #Static_1.AlarmFromID,                   
              LEN => #Static_1.AlarmLength,                 
              TINFO := #Static_1.TI_DiagnosticInterrupt,     
              AINFO := #AINFOManufacture);                   



   #SlaveType := #Static_1.TI_DiagnosticInterrupt.slv_prfl; 

   IF #SlaveType = 3 THEN      
       #Profibus_slave := 1;
       #Profinet_slave := 0;
   END_IF;

   IF #SlaveType = 8 THEN      
       #Profibus_slave := 0;
       #Profinet_slave := 1;
   END_IF;


   IF #Profinet_slave AND #Static_1.AlarmReceived AND (#AINFOManufacture.W6_interrupt_type = 16#0001) THEN
       IF (#AINFOManufacture.W26_Add_W0_format_ID = 16#7FFF) THEN
           #ALARM_1 := #AINFOManufacture.D28_AlarmWord;        
           #WARNING_1 := #AINFOManufacture.D32_WarnWord;       
           #Static_1.AlarmReceived := 0;
       END_IF;
       IF (#AINFOManufacture.W26_Add_W0_format_ID = 16#8000) THEN
           #CH_ERR_TYP := DWORD_TO_WORD(SHR(IN := (#AINFOManufacture.D32_WarnWord), N := 16)); 
           #Static_1.AlarmReceived := 0;
       END_IF;
   END_IF;


   IF #Profibus_slave AND #Static_1.AlarmReceived AND #AINFOManufacture.W2_block_length = 16#0001 THEN
       #ProfibusAlarm := #AINFOManufacture.W4_version;
       #ProfibusAlarm := SHL(IN := (#ProfibusAlarm), N := 16);
       #TempAlarm := #AINFOManufacture.W6_interrupt_type;
       #ALARM_1 := #ProfibusAlarm OR #TempAlarm;       
       #Static_1.AlarmReceived := 0;

       #ProfibusWarning := #AINFOManufacture.W12_comp_slot_num;
       #ProfibusWarning := SHL(IN := (#ProfibusWarning), N := 16);
       #TempWarning := #AINFOManufacture.W14_submodule_slot_num;
       #WARNING_1 := #ProfibusWarning OR #TempWarning;    
       #Static_1.AlarmReceived := 0;
   END_IF;


   IF #Static_1.AlarmReceived THEN
       IF #AINFOManufacture.W6_interrupt_type = 16#000C THEN
           #CH_ERR_TYP := 0;
           #ALARM_1 := 0;
           #WARNING_1 := 0;
           #Static_1.AlarmReceived := 0;
       END_IF;
   END_IF;

   IF #Static_1.AlarmReceived THEN
       IF #AINFOManufacture.W2_block_length = 2 THEN
           #CH_ERR_TYP := 0;
           #ALARM_1 := 0;
           #WARNING_1 := 0;
           #Static_1.AlarmReceived := 0;
       END_IF;
   END_IF;
END_FUNCTION_BLOCK

FUNCTION "CONVERTER" : Void   // FC1, SCL
{ S7_Optimized_Access := 'TRUE' }
VERSION : 0.1
   VAR_INPUT
      RPMDESEJADO : Int;
      CORRENTE : Int;
      FREQUENCIA : Int;
   END_VAR
   VAR_OUTPUT
      VARIADOR : Int;
      CORRENTE_SAIDA : Real;
      FREQUENCIA_SAIDA : Real;
   END_VAR
   VAR_TEMP
      FUNCTION_BLOCK : Int;
   END_VAR
BEGIN
   #VARIADOR := INT_TO_REAL (#RPMDESEJADO)*16384/1500;

   IF #VARIADOR > 16384 THEN
       #VARIADOR := 16384;


   END_IF;

   IF #VARIADOR < 0 THEN
       #VARIADOR := 0;


   END_IF;

   #CORRENTE_SAIDA := INT_TO_REAL (#CORRENTE) / 100;
   #FREQUENCIA_SAIDA := INT_TO_REAL (#FREQUENCIA) / 10;
END_FUNCTION

FUNCTION "Status" : Void   // FC2, SCL
{ S7_Optimized_Access := 'TRUE' }
VERSION : 0.1
   VAR_INPUT
      Trabalhando : Bool;
      Avaria : Bool;
      Aviso : Bool;
   END_VAR
   VAR_OUTPUT
      Status : Int;
   END_VAR
BEGIN
   IF #Trabalhando THEN
       #Status := 1;
   ELSIF #Avaria THEN
       #Status := 2;
   ELSIF #Aviso THEN
       #Status := 3;
   ELSE
       #Status := 0;
   END_IF;
END_FUNCTION

FUNCTION "VLT_PROFI_FC_BASIC" : Void   // FC300, SCL
TITLE = VLT_PROFI_FC_BASIC
{ S7_Optimized_Access := 'TRUE' }
AUTHOR : Danfoss_Drives
FAMILY : VLT
VERSION : 1.12
// Basic Operation Function Block
   VAR_INPUT
      ADR : Hw_Io;   // S7-1200/1500 requires HW Identifier. Can be found in HW configuration for the specific PPO type
      DRV_EN : Bool;   // Enable Drive. Setting the Drive in Ready to Start mode.
      RUN : Bool;   // Run/Stop drive
      REVERSE : Bool;   // Drive Reverse mode. Also set P4-10 to "both directions" to allow.
      RESET : Bool;   // Reset alarms. Only Trip, not Trip lock.
      REF_VALUE : Int;   // Reference speed 0 - 10000 = 0 - 100.00%
   END_VAR
   VAR_OUTPUT
      READY : Bool;   // Drive ready to start
      FAULT : Bool;   // Fault is present. Trip or Trip lock
      WARNING : Bool;   // Warning present
      RUNNING : Bool;   // Drive is started but not necessarily running on reference speed.
      RUN_ON_REF : Bool;   // Running on reference
      MAV : Int;   // Main Actual Value read from Drive 0 - 10000 = 0 - 100.00%
      MOTORCURRENT : Real;   // Actual motor Current
      COMM_ERR : Int;   // Result of DPRD_DAT 0=No error
   END_VAR
   VAR_TEMP
      PCDRead : Struct   // Pointer to data structure for FC data
         STW : Struct   // Status word
            BIT_00_CTRL_RDY : Bool;   // 0=Control not ready, 1=Control ready
            BIT_01_DRV_RDY : Bool;   // 0=Frequency converter, 1=Frequency converter ready
            BIT_02_COAST_RDY : Bool;   // 0=Coasting, 1=Enable
            BIT_03_TRIP : Bool;   // 0=No error, 1=Trip
            BIT_04_ERROR : Bool;   // 0=No error, 1=Error (no trip)
            BIT_05_RESERVED : Bool;   // 0=Reserved, 1=---
            BIT_06_TRIPLOCK : Bool;   // 0=No error, 1=Triplock
            BIT_07_WARNING : Bool;   // 0=No warning, 1=Warning
            BIT_08_RUNNING_REF : Bool;   // 0=Speed <> reference, 1=Speed=reference
            BIT_09_CTRL_SOURCE : Bool;   // 0=Local operation, 1=Bus control
            BIT_10_F_LIMIT_OK : Bool;   // 0=Out of frequency limit, 1=Frequency limit ok
            BIT_11_IN_OPR : Bool;   // 0=No operation, 1=In operation
            BIT_12_IN_AUTOSTART : Bool;   // 0=Frequency converter OK, 1=Stopped, autostart
            BIT_13_VOLT_MAX : Bool;   // 0=Voltage OK, 1=Voltage exceeded
            BIT_14_TORQ_MAX : Bool;   // 0=Torque OK, 1=Torque exceeded
            BIT_15_TIMER_EXD : Bool;   // 0=Timer OK, 1=Timer exceeded
         END_STRUCT;
         MAV : Int;   // Main actual value
         PCD_02 : Int;   // PCD 02
         PCD_03 : Int;   // PCD 03
         PCD_04 : Int;   // PCD 04
         PCD_05 : Int;   // PCD 05
      END_STRUCT;
      PCDWrite : Struct   // Pointer to data structure for FC data
         CTW : Struct   // Control word
            BIT_00_PRESET_REF_1 : Bool;   // 0=Reference value, 1=selection lsb
            BIT_01_PRESET_REF_2 : Bool;   // 0=Reference value, 1=selection msb
            BIT_02_DC_BRAKE_RAMP : Bool;   // 0=DC brake, 1=Ramp
            BIT_03_COAST_INV : Bool;   // 0=Coasting, 1=No coasting
            BIT_04_QSTP_RMP : Bool;   // 0=Quick stop, 1=Ramp
            BIT_05_HLD_RMP : Bool;   // 0=Hold output frequency, 1=Use ramp
            BIT_06_START : Bool;   // 0=Ramp stop, 1=Start
            BIT_07_RESET : Bool;   // 0=No function, 1=Reset
            BIT_08_JOG : Bool;   // 0=No function, 1=Jog
            BIT_09_RAMP_1_2 : Bool;   // 0=Ramp 1, 1=Ramp 2
            BIT_10_DATA_VALID : Bool;   // 0=Dont use CTW, 1= Use CTW
            BIT_11_RLY_1_ON : Bool;   // 0=Relay 01 deactived, 1=Relay 01 active
            BIT_12_RLY_2_ON : Bool;   // 0=Relay 02 deactived, 1=Relay 02 active
            BIT_13_SETUP_SEL_1 : Bool;   // 0=Parameter set-up, 1=selection lsb
            BIT_14_SETUP_SEL_2 : Bool;   // 0=Parameter set-up, 1=selection msb
            BIT_15_REVERSE : Bool;   // 0= No Reverse, 1= Reverse
         END_STRUCT;
         MRV : Int;   // Main reference value
         PCD_02 : Int;   // PCD 02
         PCD_03 : Int;   // PCD 03
         PCD_04 : Int;   // PCD 04
         PCD_05 : Int;   // PCD 05
      END_STRUCT;
      RDRaw_Data : Array[0..5] of Int;   // Data Read. PROFINET:PPO6 only, with 4 words /PROFIBUS:PPO2 only, with 6 words
      WRRaw_Data : Array[0..5] of Int;   // Data Write. PROFINET:PPO6 only, with 4 words /PROFIBUS:PPO2 only, with 6 words
      RETVAL : Int;   // Return value for DPRD and DPWR for PNET Comm. 0=no fault
      CalcSlope : Real;   // Slope of Ref. value, to convert 0-10000 into 0- 16384
      CurrentInternal : DWord;   // Internal value for current calculation
      AlwaysOn : Bool;   // Always on
      AlwaysOff : Bool;   // Always off
   END_VAR
   // // RDRaw_Data[0] : Status word
   // // RDRaw_Data[1] : Main Actual Value
   // // RDRaw_Data[2] : PCD 02
   // // RDRaw_Data[3] : PCD 03
   // // RDRaw_Data[4] : PCD 04
   // // RDRaw_Data[5] : PCD 05
   // // WRRaw_Data[0] : Control word
   // // WRRaw_Data[1] : Main Reference Value
   // // WRRaw_Data[2] : PCD 02
   // // WRRaw_Data[3] : PCD 03
   // // WRRaw_Data[4] : PCD 04
   // // WRRaw_Data[5] : PCD 05
BEGIN

   #AlwaysOff := false;
   #AlwaysOn := TRUE;

   #RETVAL := DPRD_DAT(LADDR := #ADR, RECORD => #RDRaw_Data);  
   #COMM_ERR := #RETVAL;

   #PCDRead.STW.BIT_00_CTRL_RDY := #RDRaw_Data[0].%X0;
   #PCDRead.STW.BIT_01_DRV_RDY := #RDRaw_Data[0].%X1;
   #PCDRead.STW.BIT_02_COAST_RDY := #RDRaw_Data[0].%X2;
   #PCDRead.STW.BIT_03_TRIP := #RDRaw_Data[0].%X3;
   #PCDRead.STW.BIT_04_ERROR := #RDRaw_Data[0].%X4;
   #PCDRead.STW.BIT_05_RESERVED := #RDRaw_Data[0].%X5;
   #PCDRead.STW.BIT_06_TRIPLOCK := #RDRaw_Data[0].%X6;
   #PCDRead.STW.BIT_07_WARNING := #RDRaw_Data[0].%X7;
   #PCDRead.STW.BIT_08_RUNNING_REF := #RDRaw_Data[0].%X8;
   #PCDRead.STW.BIT_09_CTRL_SOURCE := #RDRaw_Data[0].%X9;
   #PCDRead.STW.BIT_10_F_LIMIT_OK := #RDRaw_Data[0].%X10;
   #PCDRead.STW.BIT_11_IN_OPR := #RDRaw_Data[0].%X11;
   #PCDRead.STW.BIT_12_IN_AUTOSTART := #RDRaw_Data[0].%X12;
   #PCDRead.STW.BIT_13_VOLT_MAX := #RDRaw_Data[0].%X13;
   #PCDRead.STW.BIT_14_TORQ_MAX := #RDRaw_Data[0].%X14;
   #PCDRead.STW.BIT_15_TIMER_EXD := #RDRaw_Data[0].%X15;

   #PCDRead.MAV := #RDRaw_Data[1];
   #PCDRead.PCD_02 := #RDRaw_Data[2];
   #PCDRead.PCD_03 := #RDRaw_Data[3];

   IF #COMM_ERR = 0 THEN
       #CalcSlope :=LREAL_TO_REAL (10000.0 / 16384.0);
       #MAV := FLOOR_INT(#CalcSlope * #PCDRead.MAV);
   END_IF;

   IF #COMM_ERR = 0 THEN
       #CurrentInternal := DINT_TO_DWORD(#PCDRead.PCD_02); 
       #CurrentInternal := SHL_DWORD(IN := #CurrentInternal, N := 16); 
       #CurrentInternal := #CurrentInternal + DINT_TO_DWORD(#PCDRead.PCD_03); 
       #MOTORCURRENT := DINT_TO_LREAL(#CurrentInternal) / 100.0;
   END_IF;

   IF #COMM_ERR = 0 THEN
       #READY := (#PCDRead.STW.BIT_00_CTRL_RDY AND #PCDRead.STW.BIT_01_DRV_RDY AND #PCDRead.STW.BIT_02_COAST_RDY AND #PCDRead.STW.BIT_09_CTRL_SOURCE); // Drive ready to start from Fieldbus
       #RUNNING := #PCDRead.STW.BIT_11_IN_OPR; 
       #RUN_ON_REF := #PCDRead.STW.BIT_08_RUNNING_REF; 
       #WARNING := #PCDRead.STW.BIT_07_WARNING; 
       #FAULT := (#PCDRead.STW.BIT_04_ERROR OR #PCDRead.STW.BIT_03_TRIP OR #PCDRead.STW.BIT_06_TRIPLOCK); 
   ELSE
       #READY := FALSE;
       #FAULT := TRUE;
   END_IF;

   #PCDWrite.CTW.BIT_00_PRESET_REF_1 := FALSE;
   #PCDWrite.CTW.BIT_01_PRESET_REF_2 := FALSE;

   IF #DRV_EN THEN
       #PCDWrite.CTW.BIT_02_DC_BRAKE_RAMP := TRUE;
       #PCDWrite.CTW.BIT_03_COAST_INV := TRUE;
       #PCDWrite.CTW.BIT_04_QSTP_RMP := TRUE;
       #PCDWrite.CTW.BIT_05_HLD_RMP := TRUE;
   ELSE
       #PCDWrite.CTW.BIT_02_DC_BRAKE_RAMP := FALSE;
       #PCDWrite.CTW.BIT_03_COAST_INV := FALSE;
       #PCDWrite.CTW.BIT_04_QSTP_RMP := FALSE;
       #PCDWrite.CTW.BIT_05_HLD_RMP := FALSE;
   END_IF;

   #PCDWrite.CTW.BIT_06_START := FALSE;
   #PCDWrite.CTW.BIT_07_RESET := FALSE;
   #PCDWrite.CTW.BIT_08_JOG := FALSE;
   #PCDWrite.CTW.BIT_09_RAMP_1_2 := FALSE;
   #PCDWrite.CTW.BIT_10_DATA_VALID := TRUE;
   #PCDWrite.CTW.BIT_11_RLY_1_ON := FALSE;
   #PCDWrite.CTW.BIT_12_RLY_2_ON := FALSE;
   #PCDWrite.CTW.BIT_13_SETUP_SEL_1 := FALSE;
   #PCDWrite.CTW.BIT_14_SETUP_SEL_2 := FALSE;
   #PCDWrite.CTW.BIT_15_REVERSE := FALSE;

   #PCDWrite.CTW.BIT_06_START := #RUN AND NOT #FAULT; 
   #PCDWrite.CTW.BIT_15_REVERSE := #REVERSE; 
   #PCDWrite.CTW.BIT_07_RESET := #RESET; 

   IF #REF_VALUE >= 10000 THEN
       #REF_VALUE := (10000);
   END_IF;
   IF #REF_VALUE < 0 THEN
       #REF_VALUE := 0;
   END_IF;

   #WRRaw_Data[0].%X0 := #PCDWrite.CTW.BIT_00_PRESET_REF_1;
   #WRRaw_Data[0].%X1 := #PCDWrite.CTW.BIT_01_PRESET_REF_2;
   #WRRaw_Data[0].%X2 := #PCDWrite.CTW.BIT_02_DC_BRAKE_RAMP;
   #WRRaw_Data[0].%X3 := #PCDWrite.CTW.BIT_03_COAST_INV;
   #WRRaw_Data[0].%X4 := #PCDWrite.CTW.BIT_04_QSTP_RMP;
   #WRRaw_Data[0].%X5 := #PCDWrite.CTW.BIT_05_HLD_RMP;
   #WRRaw_Data[0].%X6 := #PCDWrite.CTW.BIT_06_START;
   #WRRaw_Data[0].%X7 := #PCDWrite.CTW.BIT_07_RESET;
   #WRRaw_Data[0].%X8 := #PCDWrite.CTW.BIT_08_JOG;
   #WRRaw_Data[0].%X9 := #PCDWrite.CTW.BIT_09_RAMP_1_2;
   #WRRaw_Data[0].%X10 := #PCDWrite.CTW.BIT_10_DATA_VALID;
   #WRRaw_Data[0].%X11 := #PCDWrite.CTW.BIT_11_RLY_1_ON;
   #WRRaw_Data[0].%X12 := #PCDWrite.CTW.BIT_12_RLY_2_ON;
   #WRRaw_Data[0].%X13 := #PCDWrite.CTW.BIT_13_SETUP_SEL_1;
   #WRRaw_Data[0].%X14 := #PCDWrite.CTW.BIT_14_SETUP_SEL_2;
   #WRRaw_Data[0].%X15 := #PCDWrite.CTW.BIT_15_REVERSE;

   #WRRaw_Data[2] := #PCDWrite.PCD_02;
   #WRRaw_Data[3] := #PCDWrite.PCD_03;

   IF #REF_VALUE >= 10000 THEN
       #REF_VALUE := 10000;
   END_IF;
   IF #REF_VALUE < 0 THEN
       #REF_VALUE := 0;
   END_IF;

   #CalcSlope := LREAL_TO_REAL (16384.0 / 10000.0);
   #PCDWrite.MRV := FLOOR_INT(#CalcSlope * #REF_VALUE); 
   #WRRaw_Data[1] := #PCDWrite.MRV; 

   IF #COMM_ERR = 0 THEN
       #RETVAL := DPWR_DAT(LADDR := #ADR, RECORD := #WRRaw_Data); 
       #COMM_ERR := #RETVAL;
   END_IF;


   ENO := TRUE;
END_FUNCTION

FUNCTION "VLT_PROFI_FC_FLEXIBLE" : Void   // FC301, SCL
TITLE = VLT_PROFI_FC_FLEXIBLE
{ S7_Optimized_Access := 'TRUE' }
AUTHOR : Danfoss_Drives
FAMILY : VLT
VERSION : 1.12
// Flexible Function Block
   VAR_INPUT
      ADR : Hw_Io;   // S7-1200/1500 requires HW Identifier. Can be found in HW configuration for the specific PPO type
   END_VAR
   VAR_OUTPUT
      COMM_ERR : Int;   // Result of DPRD_DAT 0=No error
   END_VAR
   VAR_IN_OUT
      PCDREAD : "PPO_READ_FCPROFILE";   // Pointer to data structure for FC data
      PCDWRITE : "PPO_WRITE_FCPROFILE";   // Pointer to data structure for FC data
   END_VAR
   VAR_TEMP
      RDRaw_Data : Array[0..9] of Int;   // Data Read. PROFINET:PPO8 only, with 10 words /PROFIBUS:PPO5 only, with 10 words
      WRRaw_Data : Array[0..9] of Int;   // Data Write. PROFINET:PPO8 only, with 10 words /PROFIBUS:PPO5 only, with 10 words
      RETVAL1 : Int;   // Internal blocks for moving data
      CalcSlope : Real;   // Slope of Ref. value, to convert 0-10000 into 0- 16384
      DUMMY : Bool;   // Internal blocks for moving data
      AlwaysOn : Bool;   // Always on
      AlwaysOff : Bool;   // Always off
   END_VAR
   // // RDRaw_Data[0] : Status word
   // // RDRaw_Data[1] : Measured Actual Value (Speed) in raw value (-16384) to (+16384)
   // // RDRaw_Data[3] : PCD 03 -Depends on Drive config.
   // // RDRaw_Data[4] : PCD 04 -Depends on Drive config.
   // // RDRaw_Data[5] : PCD 05 -Depends on Drive config.
   // // RDRaw_Data[6] : PCD 06 -Depends on Drive config.
   // // RDRaw_Data[2] : PCD 02 -Depends on Drive config.
   // // RDRaw_Data[7] : PCD 07 -Depends on Drive config.
   // // RDRaw_Data[8] : PCD 08 -Depends on Drive config.
   // // RDRaw_Data[9] : PCD 09 -Depends on Drive config.
   // // WRRaw_Data[0] : Control word
   // // WRRaw_Data[1] : Main Ref. value (Speed) in raw value. (-16384) to (+16384)
   // // WRRaw_Data[2] : PCD 02 -Depends on Drive config.
   // // WRRaw_Data[3] : PCD 03 -Depends on Drive config.
   // // WRRaw_Data[4] : PCD 04 -Depends on Drive config.
   // // WRRaw_Data[5] : PCD 05 -Depends on Drive config.
   // // WRRaw_Data[6] : PCD 06 -Depends on Drive config.
   // // WRRaw_Data[7] : PCD 07 -Depends on Drive config.
   // // WRRaw_Data[8] : PCD 08 -Depends on Drive config.
   // // WRRaw_Data[9] : PCD 09 -Depends on Drive config.
BEGIN

   #AlwaysOff := FALSE;
   #AlwaysOn := TRUE;

   #RETVAL1 := DPRD_DAT(LADDR := #ADR, RECORD => #RDRaw_Data); 
   #COMM_ERR := #RETVAL1;

   #PCDREAD.STW.BIT_00_CTRL_RDY := #RDRaw_Data[0].%X0;
   #PCDREAD.STW.BIT_01_DRV_RDY := #RDRaw_Data[0].%X1;
   #PCDREAD.STW.BIT_02_COAST_RDY := #RDRaw_Data[0].%X2;
   #PCDREAD.STW.BIT_03_TRIP := #RDRaw_Data[0].%X3;
   #PCDREAD.STW.BIT_04_ERROR := #RDRaw_Data[0].%X4;
   #PCDREAD.STW.BIT_05_RESERVED := #RDRaw_Data[0].%X5;
   #PCDREAD.STW.BIT_06_TRIPLOCK := #RDRaw_Data[0].%X6;
   #PCDREAD.STW.BIT_07_WARNING := #RDRaw_Data[0].%X7;
   #PCDREAD.STW.BIT_08_RUNNING_REF := #RDRaw_Data[0].%X8;
   #PCDREAD.STW.BIT_09_CTRL_SOURCE := #RDRaw_Data[0].%X9;
   #PCDREAD.STW.BIT_10_F_LIMIT_OK := #RDRaw_Data[0].%X10;
   #PCDREAD.STW.BIT_11_IN_OPR := #RDRaw_Data[0].%X11;
   #PCDREAD.STW.BIT_12_IN_AUTOSTART := #RDRaw_Data[0].%X12;
   #PCDREAD.STW.BIT_13_VOLT_MAX := #RDRaw_Data[0].%X13;
   #PCDREAD.STW.BIT_14_TORQ_MAX := #RDRaw_Data[0].%X14;
   #PCDREAD.STW.BIT_15_TIMER_EXD := #RDRaw_Data[0].%X15;

   #PCDREAD.MAV := #RDRaw_Data[1];
   #PCDREAD.PCD_02 := #RDRaw_Data[2];
   #PCDREAD.PCD_03 := #RDRaw_Data[3];
   #PCDREAD.PCD_04 := #RDRaw_Data[4];
   #PCDREAD.PCD_05 := #RDRaw_Data[5];
   #PCDREAD.PCD_06 := #RDRaw_Data[6];
   #PCDREAD.PCD_07 := #RDRaw_Data[7];
   #PCDREAD.PCD_08 := #RDRaw_Data[8];
   #PCDREAD.PCD_09 := #RDRaw_Data[9];

   #WRRaw_Data[0].%X0 := #PCDWRITE.CTW.BIT_00_PRESET_REF_1;
   #WRRaw_Data[0].%X1 := #PCDWRITE.CTW.BIT_01_PRESET_REF_2;
   #WRRaw_Data[0].%X2 := #PCDWRITE.CTW.BIT_02_DC_BRAKE_RAMP;
   #WRRaw_Data[0].%X3 := #PCDWRITE.CTW.BIT_03_COAST_INV;
   #WRRaw_Data[0].%X4 := #PCDWRITE.CTW.BIT_04_QSTP_RMP;
   #WRRaw_Data[0].%X5 := #PCDWRITE.CTW.BIT_05_HLD_RMP;
   #WRRaw_Data[0].%X6 := #PCDWRITE.CTW.BIT_06_START;
   #WRRaw_Data[0].%X7 := #PCDWRITE.CTW.BIT_07_RESET;
   #WRRaw_Data[0].%X8 := #PCDWRITE.CTW.BIT_08_JOG;
   #WRRaw_Data[0].%X9 := #PCDWRITE.CTW.BIT_09_RAMP_1_2;
   #WRRaw_Data[0].%X10 := #PCDWRITE.CTW.BIT_10_DATA_VALID;
   #WRRaw_Data[0].%X11 := #PCDWRITE.CTW.BIT_11_RLY_1_ON;
   #WRRaw_Data[0].%X12 := #PCDWRITE.CTW.BIT_12_RLY_2_ON;
   #WRRaw_Data[0].%X13 := #PCDWRITE.CTW.BIT_13_SETUP_SEL_1;
   #WRRaw_Data[0].%X14 := #PCDWRITE.CTW.BIT_14_SETUP_SEL_2;
   #WRRaw_Data[0].%X15 := #PCDWRITE.CTW.BIT_15_REVERSE;

   #WRRaw_Data[1] := #PCDWRITE.REF_VALUE;
   #WRRaw_Data[2] := #PCDWRITE.PCD_02;
   #WRRaw_Data[3] := #PCDWRITE.PCD_03;
   #WRRaw_Data[4] := #PCDWRITE.PCD_04;
   #WRRaw_Data[5] := #PCDWRITE.PCD_05;
   #WRRaw_Data[6] := #PCDWRITE.PCD_06;
   #WRRaw_Data[7] := #PCDWRITE.PCD_07;
   #WRRaw_Data[8] := #PCDWRITE.PCD_08;
   #WRRaw_Data[9] := #PCDWRITE.PCD_09;


   IF #RETVAL1 = 0 THEN
       #RETVAL1 := DPWR_DAT(LADDR := #ADR, RECORD := #WRRaw_Data); // Write Raw Data 
       #COMM_ERR := #RETVAL1;
   END_IF;

   ENO := TRUE;
END_FUNCTION

(* ===== HMI "HMI_RT_1" =====
system functions are stored by id; their names below are inferred from use
connection "Connection_1": ETHERNET, SMART_S7_1200_OMS
connection "HMI_Connection_1": ETHERNET, SMART_S7_1200_OMS

HMI tags "Default tag table"
   "Velocidade_Desejada" : Int = PLC Tag_3 AT %MW300, 1 s
   "Start_Driver" : Bool = PLC START_FLEXIBLE_CTRL_DUT1 AT %M44.0, 1 s
   "Reset_Driver" : Bool = PLC RESET_DUT_FLEXIBLE_CTRL_DUT1 AT %M45.2, 1 s
   "Jog" : Bool = PLC JOG_DUT1 AT %M45.3, 1 s
   "Reversao" : Bool = PLC REVERSE_FLEXIBLE_CTRl_DUT1 AT %M48.1, 1 s
   "Ready" : Bool = PLC READ_FLEXIBLE_CTRL_DUT1 AT %M48.2, 1 s
   "Fault" : Bool = PLC FALUT_FLEXIBLE_CTRL_DUT1 AT %M48.3, 1 s
   "Warning" : Bool = PLC WARNING_FLEXIBLE_CTRL_DUT1 AT %M48.4, 1 s
   "Running" : Bool = PLC RUNNING_FLEXIBLE_CTRL_DUT1 AT %M48.6, 1 s
   "Corrente" : Real = PLC Tag_15 AT %MD314, 1 s
   "Status_Motor" : Int = PLC Tag_5 AT %MW306, 100 ms
   "Frequencia" : Real = PLC Tag_16 AT %MD318, 1 s

HMI tags "Tag table_1"
   "HMI_Tag_1(1)" : Int, internal

graphic list "Graphic_list_1": 1 'Graphic_3'; 2 'Graphic_6'; 3 'Graphic_7'; 0 'Graphic_5'

Template "Template_1" 800x480
   Button "Exit" at 714,429 size 71x50; TextOff 'Exit'; PictureOff "ExitRuntime_KTP700_Basic_PN_TR"; PictureOn "ExitRuntime_KTP700_Basic_PN_TR"
      on Release: StopRuntime(0)
   Button "Log on" at 614,429 size 71x50; TextOff 'Log on'; PictureOff "Login_KTP700_Basic_PN_TR"; PictureOn "Login_KTP700_Basic_PN_TR"
      on Release: function_a2a04561()
   Button "Template_Button" at 514,429 size 71x50; TextOff 'Text'
   Button "Template_Button_1" at 414,429 size 71x50; TextOff 'Text'
   Button "Template_Button_2" at 314,429 size 71x50; TextOff 'Text'
   Button "Template_Button_3" at 214,429 size 71x50; TextOff 'Text'
   Button "Alarms" at 114,429 size 71x50; TextOff 'Alarms'; PictureOff "AlarmDisplay_KTP700_Basic_PN_TR"; PictureOn "AlarmDisplay_KTP700_Basic_PN_TR"
      on Release: function_ef3f5d25("Alarm window_Unacknowledged", -1)
   Button "Start screen" at 14,429 size 71x50; TextOff 'Start screen'; PictureOff "NavigateHome_KTP700_Basic_PN_TR"; PictureOn "NavigateHome_KTP700_Basic_PN_TR"
      on Release: ActivateScreen("Root screen", 0)
   DateTimeField "HmiScreenItemData" at 695,25 size 105x25
   DateTimeField "HmiScreenItemData_1" at 695,0 size 105x25

screen "Root screen" 800x480, template "Template_1"
   GraphicIOField "Graphic I/O field_1" at 211,166 size 206x145; PictureList "Graphic_list_1"
      ProcessValue <- "Status_Motor"
   Button "Button_1" at 39,92 size 130x48; TextOff 'Start'
      on Release: InvertBit("Start_Driver")
      Appearance <- "Start_Driver"
   Button "Button_2" at 39,149 size 130x48; TextOff 'Reset'
   Button "Button_3" at 39,206 size 130x48; TextOff 'Reversao'
      on Release: InvertBit("Reversao")
      Appearance <- "Reversao"
   IOField "I/O field_1" at 37,326 size 132x60; FormatPattern 99999; Unit  RPM
      ProcessValue <- "Velocidade_Desejada"
   TextField "Text field_1" at 234,101 size 126x23; Text 'Corrente Atual'
   IOField "I/O field_3" at 229,129 size 136x37; FormatPattern 99.99; Unit  A
      ProcessValue <- "Corrente"
   Button "Button_4" at 39,263 size 130x48; TextOff 'Jog'
      on Release: InvertBit("Jog")
      Appearance <- "Jog"
   TrendView "Trend view_1" at 421,92 size 343x296
   TextField "Text field_2" at 234,357 size 143x23; Text 'Frequencia Atual'
   IOField "I/O field_2" at 229,318 size 136x37; FormatPattern 99.99; Unit  HZ
      ProcessValue <- "Frequencia"
*)